// TIA Portal V16 program export: 0 tag tables, 14 data types, 2 data blocks, 1 code blocks (in call order from the OBs), 2 instance data blocks

TYPE "ConfigIF_MPLC_to_Plant"
// stored: IsFailsafeCompliant false
   STRUCT
      Spare_1 { ExternalAccessible := 'False'; ExternalVisible := 'False'; ExternalWritable := 'False'} : Word;   // Machine Features (refer to the Standard Machine Configuration Data)
      Machine_Product_ID { ExternalAccessible := 'False'; ExternalVisible := 'False'; ExternalWritable := 'False'} : Byte;   // Machine Product ID (refer to the Standard Machine Configuration Data)
      Machine_SortFraction { ExternalAccessible := 'False'; ExternalVisible := 'False'; ExternalWritable := 'False'} : Byte;   // Machine Sort Fraction (refer to the Standard Machine Configuration Data)
      Machine_Function { ExternalAccessible := 'False'; ExternalVisible := 'False'; ExternalWritable := 'False'} : Byte;   // Machine Function (refer to the Standard Machine Configuration Data)
      Machine_Cluster_ID { ExternalAccessible := 'False'; ExternalVisible := 'False'; ExternalWritable := 'False'} : Byte;   // Machine Cluster number (0-255)
      Machine_Cluster_Configuration { ExternalAccessible := 'False'; ExternalVisible := 'False'; ExternalWritable := 'False'} : Word;   // Machine Cluster Configuration (refer to the Standard Machine Configuration Data)
      PCS_PrimaryProtocol { ExternalAccessible := 'False'; ExternalVisible := 'False'; ExternalWritable := 'False'} : Byte;   // Primary Plant communication Protocol (Refer to Standard Machine Configuration Document)
      PCS_SecondaryProtocol { ExternalAccessible := 'False'; ExternalVisible := 'False'; ExternalWritable := 'False'} : Byte;   // Secondary Plant communication Protocol (Refer to Standard Machine Configuration Document)
      Hardware_Configuration_ID { ExternalAccessible := 'False'; ExternalVisible := 'False'; ExternalWritable := 'False'} : Byte;   // Machine PLC hardware configuration option (0-255)
      OPC_UA_ControlClient { ExternalAccessible := 'False'; ExternalVisible := 'False'; ExternalWritable := 'False'} : Bool;   // 0= Control Client Disabled; 1=Control Client Enabled
      OPC_UA_ViewClient_1 { ExternalAccessible := 'False'; ExternalVisible := 'False'; ExternalWritable := 'False'} : Bool;   // 0= View Client 1 Disabled; 1=View Client 1 Enabled
      OPC_UA_ViewClient_2 { ExternalAccessible := 'False'; ExternalVisible := 'False'; ExternalWritable := 'False'} : Bool;   // 0= View Client 2 Disabled; 1=View Client 2 Enabled
      OPC_UA_ViewClient_3 { ExternalAccessible := 'False'; ExternalVisible := 'False'; ExternalWritable := 'False'} : Bool;   // 0= View Client 3 Disabled; 1=View Client 3 Enabled
      Spare11_4 { ExternalAccessible := 'False'; ExternalVisible := 'False'; ExternalWritable := 'False'} : Bool;   // Reserved spare
      Spare11_5 { ExternalAccessible := 'False'; ExternalVisible := 'False'; ExternalWritable := 'False'} : Bool;   // Reserved spare
      Spare11_6 { ExternalAccessible := 'False'; ExternalVisible := 'False'; ExternalWritable := 'False'} : Bool;   // Reserved spare
      Spare11_7 { ExternalAccessible := 'False'; ExternalVisible := 'False'; ExternalWritable := 'False'} : Bool;   // Reserved spare
      Machine_IP_Address { ExternalAccessible := 'False'; ExternalVisible := 'False'; ExternalWritable := 'False'} : Array[1..4] of Byte;   // Machine PLC IP address (xx-xx-xx-xx)
      Machine_TCP_Port { ExternalAccessible := 'False'; ExternalVisible := 'False'; ExternalWritable := 'False'} : Int;   // Machine PLC TCP port number (2010-5000)
      Machine_TSAP { ExternalAccessible := 'False'; ExternalVisible := 'False'; ExternalWritable := 'False'} : Array[1..16] of Byte;   // Machine PLC TSAP (string containing Machine to 16 x ASCII characters)
      Machine_MAC_Address { ExternalAccessible := 'False'; ExternalVisible := 'False'; ExternalWritable := 'False'} : Array[0..5] of Byte;   // Machine PLC MAC address (xx-xx-xx-xx-xx-xx)
      Plant_Connection_ID { ExternalAccessible := 'False'; ExternalVisible := 'False'; ExternalWritable := 'False'} : Int;   // Plant PLC connection reference (1-65535)
      Spare { ExternalAccessible := 'False'; ExternalVisible := 'False'; ExternalWritable := 'False'} : Int;   // Reserved spare
      NTP_Server_IP_Address { ExternalAccessible := 'False'; ExternalVisible := 'False'; ExternalWritable := 'False'} : Array[1..4] of Byte;   // NTP Time Server Address (xx-xx-xx-xx)
      Last_PCS_Config_Hours { ExternalAccessible := 'False'; ExternalVisible := 'False'; ExternalWritable := 'False'} : Byte;   // Last configuration date/time recorded on the PLC after PCS config request from OTI or Plant. OTI/SCADA username transferred by PLC (depending on the config source)
      Last_PCS_Config_Minutes { ExternalAccessible := 'False'; ExternalVisible := 'False'; ExternalWritable := 'False'} : Byte;   // As above
      Last_PCS_Config_Century { ExternalAccessible := 'False'; ExternalVisible := 'False'; ExternalWritable := 'False'} : Byte;   // As above
      Last_PCS_Config_Year { ExternalAccessible := 'False'; ExternalVisible := 'False'; ExternalWritable := 'False'} : Byte;   // As above
      Last_PCS_Config_Month { ExternalAccessible := 'False'; ExternalVisible := 'False'; ExternalWritable := 'False'} : Byte;   // As above
      Last_PCS_Config_Day { ExternalAccessible := 'False'; ExternalVisible := 'False'; ExternalWritable := 'False'} : Byte;   // As above
      UserName { ExternalAccessible := 'False'; ExternalVisible := 'False'; ExternalWritable := 'False'} : Array[0..7] of Byte;   // Name of user (SCADA or OTI), who performed PCS configuration
      PCS_Config_Source { ExternalAccessible := 'False'; ExternalVisible := 'False'; ExternalWritable := 'False'} : Byte;   // PCS Configuration source: 0 - None; 1 - OTI; 2 - Plant
      OPC_UA_ControlClient_Active { ExternalAccessible := 'False'; ExternalVisible := 'False'; ExternalWritable := 'False'} : Bool;   // 1=OPC-UA ControlClient Active; 0=OPC-UA ControlClient Inactive
      OPC_UA_ViewClient_1_Active { ExternalAccessible := 'False'; ExternalVisible := 'False'; ExternalWritable := 'False'} : Bool;   // 1=OPC-UA ViewClient_1 Active; 0=OPC-UA ViewClient_1 Inactive
      OPC_UA_ViewClient_2_Active { ExternalAccessible := 'False'; ExternalVisible := 'False'; ExternalWritable := 'False'} : Bool;   // 1=OPC-UA ViewClient_2 Active; 0=OPC-UA ViewClient_2 Inactive
      OPC_UA_ViewClient_3_Active { ExternalAccessible := 'False'; ExternalVisible := 'False'; ExternalWritable := 'False'} : Bool;   // 1=OPC-UA ViewClient_3 Active; 0=OPC-UA ViewClient_3 Inactive
      Spare63_4 { ExternalAccessible := 'False'; ExternalVisible := 'False'; ExternalWritable := 'False'} : Bool;   // Reserved spare
      Spare63_5 { ExternalAccessible := 'False'; ExternalVisible := 'False'; ExternalWritable := 'False'} : Bool;   // Reserved spare
      Primary_Protocol_Comms_OK { ExternalAccessible := 'False'; ExternalVisible := 'False'; ExternalWritable := 'False'} : Bool;   // Plant Control Network Communication Status (0=Error; 1=OK)
      Secondary_Protocol_Comms_OK { ExternalAccessible := 'False'; ExternalVisible := 'False'; ExternalWritable := 'False'} : Bool;   // Plant SMachineervision Network Communication Status (0=Error; 1=OK)
      OPC_UA_PortNumber { ExternalAccessible := 'False'; ExternalVisible := 'False'; ExternalWritable := 'False'} : UInt;   // Machine- configured OPC-UA port
      Profibus_Address { ExternalAccessible := 'False'; ExternalVisible := 'False'; ExternalWritable := 'False'} : Byte;   // Machine- configured Profibus Address
      Spare67 { ExternalAccessible := 'False'; ExternalVisible := 'False'; ExternalWritable := 'False'} : Byte;   // Reserved spare
      Spare68 { ExternalAccessible := 'False'; ExternalVisible := 'False'; ExternalWritable := 'False'} : Byte;   // Reserved spare
      Spare69 { ExternalAccessible := 'False'; ExternalVisible := 'False'; ExternalWritable := 'False'} : Byte;   // Reserved spare
      Spare70 { ExternalAccessible := 'False'; ExternalVisible := 'False'; ExternalWritable := 'False'} : Byte;   // Reserved spare
      Spare71 { ExternalAccessible := 'False'; ExternalVisible := 'False'; ExternalWritable := 'False'} : Byte;   // Reserved spare
      Spare72 { ExternalAccessible := 'False'; ExternalVisible := 'False'; ExternalWritable := 'False'} : Byte;   // Reserved spare
      Spare73 { ExternalAccessible := 'False'; ExternalVisible := 'False'; ExternalWritable := 'False'} : Byte;   // Reserved spare
      Spare74 { ExternalAccessible := 'False'; ExternalVisible := 'False'; ExternalWritable := 'False'} : Byte;   // Reserved spare
      Spare75 { ExternalAccessible := 'False'; ExternalVisible := 'False'; ExternalWritable := 'False'} : Byte;   // Reserved spare
      Spare76 { ExternalAccessible := 'False'; ExternalVisible := 'False'; ExternalWritable := 'False'} : Byte;   // Reserved spare
      Spare77 { ExternalAccessible := 'False'; ExternalVisible := 'False'; ExternalWritable := 'False'} : Byte;   // Reserved spare
      Spare78 { ExternalAccessible := 'False'; ExternalVisible := 'False'; ExternalWritable := 'False'} : Byte;   // Reserved spare
      Spare79 { ExternalAccessible := 'False'; ExternalVisible := 'False'; ExternalWritable := 'False'} : Byte;   // Reserved spare
      Spare80 { ExternalAccessible := 'False'; ExternalVisible := 'False'; ExternalWritable := 'False'} : Byte;   // Reserved spare
      Spare81 { ExternalAccessible := 'False'; ExternalVisible := 'False'; ExternalWritable := 'False'} : Byte;   // Reserved spare
      Spare82 { ExternalAccessible := 'False'; ExternalVisible := 'False'; ExternalWritable := 'False'} : Byte;   // Reserved spare
      Spare83 { ExternalAccessible := 'False'; ExternalVisible := 'False'; ExternalWritable := 'False'} : Byte;   // Reserved spare
      Spare84 { ExternalAccessible := 'False'; ExternalVisible := 'False'; ExternalWritable := 'False'} : Byte;   // Reserved spare
      Spare85 { ExternalAccessible := 'False'; ExternalVisible := 'False'; ExternalWritable := 'False'} : Byte;   // Reserved spare
      Spare86 { ExternalAccessible := 'False'; ExternalVisible := 'False'; ExternalWritable := 'False'} : Byte;   // Reserved spare
      Spare87 { ExternalAccessible := 'False'; ExternalVisible := 'False'; ExternalWritable := 'False'} : Byte;   // Reserved spare
      Spare88 { ExternalAccessible := 'False'; ExternalVisible := 'False'; ExternalWritable := 'False'} : Byte;   // Reserved spare
      Spare89 { ExternalAccessible := 'False'; ExternalVisible := 'False'; ExternalWritable := 'False'} : Byte;   // Reserved spare
      Machine_Features { ExternalAccessible := 'False'; ExternalVisible := 'False'; ExternalWritable := 'False'} : DWord;   // Machine Features (refer to the Standard Machine Configuration Data)
      Machine_Features_Mask { ExternalAccessible := 'False'; ExternalVisible := 'False'; ExternalWritable := 'False'} : DWord;   // Machine Features Mask (refer to the Standard Machine Configuration Data)
      OTI_CheckCycle_Override_Control_State { ExternalAccessible := 'False'; ExternalVisible := 'False'; ExternalWritable := 'False'} : Bool;   // 1 = 'Override Checkercycle' control on OTI Disabled
      OTI_Configuration_Control_Status { ExternalAccessible := 'False'; ExternalVisible := 'False'; ExternalWritable := 'False'} : Bool;   // 1 = OTI PCS Configuration Machinedate button disabled
      OTI_PCS_Config { ExternalAccessible := 'False'; ExternalVisible := 'False'; ExternalWritable := 'False'} : Bool;   // Configuration pulse from OTI (pulsed for 1sec)
      OTI_Authentication_Mode { ExternalAccessible := 'False'; ExternalVisible := 'False'; ExternalWritable := 'False'} : Bool;   // Machine user authentication mode (0=password; 1= biometrics)
      Machine_Init { ExternalAccessible := 'False'; ExternalVisible := 'False'; ExternalWritable := 'False'} : Bool;   // PLC IP Address /HW Config Machinedate pulse (pulsed for 1sec)
      OTI_Ej_Sense_Feedback_Control_State { ExternalAccessible := 'False'; ExternalVisible := 'False'; ExternalWritable := 'False'} : Bool;   // 1 = 'Override Ejector Sense Feedback Alarms' on OTI disabled
      Spare98_6 { ExternalAccessible := 'False'; ExternalVisible := 'False'; ExternalWritable := 'False'} : Bool;   // Reserved spare
      TimeSync_Source { ExternalAccessible := 'False'; ExternalVisible := 'False'; ExternalWritable := 'False'} : Bool;   // Time Synchronization Source (0=NTP Server; 1= Interface DB)
      Spare99_0 { ExternalAccessible := 'False'; ExternalVisible := 'False'; ExternalWritable := 'False'} : Bool;   // Reserved spare
      Spare99_1 { ExternalAccessible := 'False'; ExternalVisible := 'False'; ExternalWritable := 'False'} : Bool;   // Reserved spare
      Spare99_2 { ExternalAccessible := 'False'; ExternalVisible := 'False'; ExternalWritable := 'False'} : Bool;   // Reserved spare
      Spare99_3 { ExternalAccessible := 'False'; ExternalVisible := 'False'; ExternalWritable := 'False'} : Bool;   // Reserved spare
      Spare99_4 { ExternalAccessible := 'False'; ExternalVisible := 'False'; ExternalWritable := 'False'} : Bool;   // Reserved spare
      Spare99_5 { ExternalAccessible := 'False'; ExternalVisible := 'False'; ExternalWritable := 'False'} : Bool;   // Reserved spare
      Spare99_6 { ExternalAccessible := 'False'; ExternalVisible := 'False'; ExternalWritable := 'False'} : Bool;   // Reserved spare
      PCS_Config_Machinedate_Done { ExternalAccessible := 'False'; ExternalVisible := 'False'; ExternalWritable := 'False'} : Bool;   // 1 sec Confirmation pulse – configuration date, time and username recorded in the event log
   END_STRUCT;
END_TYPE

TYPE "ConfigIF_Plant_to_MPLC"
// stored: IsFailsafeCompliant false
   STRUCT
      Plant_ID { ExternalAccessible := 'False'; ExternalVisible := 'False'; ExternalWritable := 'False'} : Byte;   // Plant location code (Refer to Standard Machine Configuration Document)
      Area_ID { ExternalAccessible := 'False'; ExternalVisible := 'False'; ExternalWritable := 'False'} : Byte;   // Plant Area code (Refer to Standard Machine Configuration Document)
      Spare2 { ExternalAccessible := 'False'; ExternalVisible := 'False'; ExternalWritable := 'False'} : Byte;   // Reserved spare
      Machine_SortFraction { ExternalAccessible := 'False'; ExternalVisible := 'False'; ExternalWritable := 'False'} : Byte;   // Machine Sort Fraction (Refer to Standard Machine Configuration Document)
      Machine_Function { ExternalAccessible := 'False'; ExternalVisible := 'False'; ExternalWritable := 'False'} : Byte;   // Machine Function (Refer to Standard Machine Configuration Document)
      Machine_Cluster_ID { ExternalAccessible := 'False'; ExternalVisible := 'False'; ExternalWritable := 'False'} : Byte;   // Machine Cluster number (0-255)
      Machine_Cluster_Configuration { ExternalAccessible := 'False'; ExternalVisible := 'False'; ExternalWritable := 'False'} : UInt;   // Machine Cluster Configuration (Maximum of 4 Machine Functions)
      Station_Name { ExternalAccessible := 'False'; ExternalVisible := 'False'; ExternalWritable := 'False'} : Array[0..15] of Byte;   // Machine Station name (string containing 16 x ASCII characters)
      PCS_Type { ExternalAccessible := 'False'; ExternalVisible := 'False'; ExternalWritable := 'False'} : Byte;   // SCADA/Plant control system type
      PCS_SecondaryProtocol { ExternalAccessible := 'False'; ExternalVisible := 'False'; ExternalWritable := 'False'} : Byte;   // Secondary Plant communication Protocol (Refer to Standard Machine Configuration Document)
      Plant_PLC_Type { ExternalAccessible := 'False'; ExternalVisible := 'False'; ExternalWritable := 'False'} : Byte;   // Plant PLC type and model
      OPCUA_ControlClient { ExternalAccessible := 'False'; ExternalVisible := 'False'; ExternalWritable := 'False'} : Bool;   // 0= Control Client Disabled; 1=Control Client Enabled
      OPCUA_ViewClient_1 { ExternalAccessible := 'False'; ExternalVisible := 'False'; ExternalWritable := 'False'} : Bool;   // 0= View Client 1 Disabled; 1=View Client 1 Enabled
      OPCUA_ViewClient_2 { ExternalAccessible := 'False'; ExternalVisible := 'False'; ExternalWritable := 'False'} : Bool;   // 0= View Client 2 Disabled; 1=View Client 2 Enabled
      OPCUA_ViewClient_3 { ExternalAccessible := 'False'; ExternalVisible := 'False'; ExternalWritable := 'False'} : Bool;   // 0= View Client 3 Disabled; 1=View Client 3 Enabled
      Spare27_4 { ExternalAccessible := 'False'; ExternalVisible := 'False'; ExternalWritable := 'False'} : Bool;   // Reserved spare
      Spare27_5 { ExternalAccessible := 'False'; ExternalVisible := 'False'; ExternalWritable := 'False'} : Bool;   // Reserved spare
      Spare27_6 { ExternalAccessible := 'False'; ExternalVisible := 'False'; ExternalWritable := 'False'} : Bool;   // Reserved spare
      Spare27_7 { ExternalAccessible := 'False'; ExternalVisible := 'False'; ExternalWritable := 'False'} : Bool;   // Reserved spare
      Spare28_4 { ExternalAccessible := 'False'; ExternalVisible := 'False'; ExternalWritable := 'False'} : DWord;   // Reserved spare
      Spare32_4 { ExternalAccessible := 'False'; ExternalVisible := 'False'; ExternalWritable := 'False'} : DWord;   // Reserved spare
      Spare36_4 { ExternalAccessible := 'False'; ExternalVisible := 'False'; ExternalWritable := 'False'} : DWord;   // Reserved spare
      Plant_IP_Address { ExternalAccessible := 'False'; ExternalVisible := 'False'; ExternalWritable := 'False'} : Array[1..4] of Byte;   // Plant PLC IP address (xx-xx-xx-xx)
      Machine_Port_Number { ExternalAccessible := 'False'; ExternalVisible := 'False'; ExternalWritable := 'False'} : UInt;   // Machine PLC TCP port number (2010-5000)
      Plant_Port_Number { ExternalAccessible := 'False'; ExternalVisible := 'False'; ExternalWritable := 'False'} : UInt;   // Plant PLC TCP port number (2010-5000)
      Machine_TSAP { ExternalAccessible := 'False'; ExternalVisible := 'False'; ExternalWritable := 'False'} : Array[1..16] of Byte;   // Machine PLC TSAP (string containing Machine to 16 x ASCII characters)
      Plant_TSAP { ExternalAccessible := 'False'; ExternalVisible := 'False'; ExternalWritable := 'False'} : Array[1..16] of Byte;   // Plant PLC TSAP (string containing Machine to 16 x ASCII characters)
      Spare80_4 { ExternalAccessible := 'False'; ExternalVisible := 'False'; ExternalWritable := 'False'} : DWord;   // Reserved spare
      Spare84_2 { ExternalAccessible := 'False'; ExternalVisible := 'False'; ExternalWritable := 'False'} : Word;   // Reserved spare
      Plant_MAC_Address { ExternalAccessible := 'False'; ExternalVisible := 'False'; ExternalWritable := 'False'} : Array[0..5] of Byte;   // Plant PLC MAC address (xx-xx-xx-xx)
      PCS_Connection_ID { ExternalAccessible := 'False'; ExternalVisible := 'False'; ExternalWritable := 'False'} : UInt;   // Plant PLC connection reference (1-65535)
      NTP_Server_IP_Address { ExternalAccessible := 'False'; ExternalVisible := 'False'; ExternalWritable := 'False'} : Array[1..4] of Byte;   // NTP time server address (xx-xx-xx-xx)
      UserName { ExternalAccessible := 'False'; ExternalVisible := 'False'; ExternalWritable := 'False'} : Array[0..7] of Byte;   // SCADA login username (Machine to 8 ASCII characters)
      DataServer_IP_Address { ExternalAccessible := 'False'; ExternalVisible := 'False'; ExternalWritable := 'False'} : Array[1..4] of Byte;   // Shared Data Server IP Address (xx-xx-xx-xx)
      DataServer_Subnet_Mask { ExternalAccessible := 'False'; ExternalVisible := 'False'; ExternalWritable := 'False'} : Array[1..4] of Byte;   // Shared Data Server Subnet Mask (xx-xx-xx-xx)
      DNS_Server_Address { ExternalAccessible := 'False'; ExternalVisible := 'False'; ExternalWritable := 'False'} : Array[1..4] of Byte;   // Domain Name System IP Address (xx-xx-xx-xx)
      Spare118 { ExternalAccessible := 'False'; ExternalVisible := 'False'; ExternalWritable := 'False'} : Byte;   // Reserved spare
      Spare119 { ExternalAccessible := 'False'; ExternalVisible := 'False'; ExternalWritable := 'False'} : Byte;   // Reserved spare
      Spare120 { ExternalAccessible := 'False'; ExternalVisible := 'False'; ExternalWritable := 'False'} : Byte;   // Reserved spare
      Spare121 { ExternalAccessible := 'False'; ExternalVisible := 'False'; ExternalWritable := 'False'} : Byte;   // Reserved spare
      Spare122 { ExternalAccessible := 'False'; ExternalVisible := 'False'; ExternalWritable := 'False'} : Byte;   // Reserved spare
      Spare123 { ExternalAccessible := 'False'; ExternalVisible := 'False'; ExternalWritable := 'False'} : Byte;   // Reserved spare
      Spare124 { ExternalAccessible := 'False'; ExternalVisible := 'False'; ExternalWritable := 'False'} : Byte;   // Reserved spare
      Spare125 { ExternalAccessible := 'False'; ExternalVisible := 'False'; ExternalWritable := 'False'} : Byte;   // Reserved spare
      Spare126 { ExternalAccessible := 'False'; ExternalVisible := 'False'; ExternalWritable := 'False'} : Byte;   // Reserved spare
      Spare127 { ExternalAccessible := 'False'; ExternalVisible := 'False'; ExternalWritable := 'False'} : Byte;   // Reserved spare
      Spare128 { ExternalAccessible := 'False'; ExternalVisible := 'False'; ExternalWritable := 'False'} : Byte;   // Reserved spare
      Spare129 { ExternalAccessible := 'False'; ExternalVisible := 'False'; ExternalWritable := 'False'} : Byte;   // Reserved spare
      Spare130 { ExternalAccessible := 'False'; ExternalVisible := 'False'; ExternalWritable := 'False'} : Byte;   // Reserved spare
      Spare131 { ExternalAccessible := 'False'; ExternalVisible := 'False'; ExternalWritable := 'False'} : Byte;   // Reserved spare
      Spare132 { ExternalAccessible := 'False'; ExternalVisible := 'False'; ExternalWritable := 'False'} : Byte;   // Reserved spare
      Spare133 { ExternalAccessible := 'False'; ExternalVisible := 'False'; ExternalWritable := 'False'} : Byte;   // Reserved spare
      Spare134 { ExternalAccessible := 'False'; ExternalVisible := 'False'; ExternalWritable := 'False'} : Byte;   // Reserved spare
      Spare135 { ExternalAccessible := 'False'; ExternalVisible := 'False'; ExternalWritable := 'False'} : Byte;   // Reserved spare
      Spare136 { ExternalAccessible := 'False'; ExternalVisible := 'False'; ExternalWritable := 'False'} : Byte;   // Reserved spare
      Spare137 { ExternalAccessible := 'False'; ExternalVisible := 'False'; ExternalWritable := 'False'} : Byte;   // Reserved spare
      Spare138 { ExternalAccessible := 'False'; ExternalVisible := 'False'; ExternalWritable := 'False'} : Byte;   // Reserved spare
      Spare139 { ExternalAccessible := 'False'; ExternalVisible := 'False'; ExternalWritable := 'False'} : Byte;   // Reserved spare
      Spare140 { ExternalAccessible := 'False'; ExternalVisible := 'False'; ExternalWritable := 'False'} : Byte;   // Reserved spare
      Spare141 { ExternalAccessible := 'False'; ExternalVisible := 'False'; ExternalWritable := 'False'} : Byte;   // Reserved spare
      Spare142 { ExternalAccessible := 'False'; ExternalVisible := 'False'; ExternalWritable := 'False'} : Byte;   // Reserved spare
      Spare143 { ExternalAccessible := 'False'; ExternalVisible := 'False'; ExternalWritable := 'False'} : Byte;   // Reserved spare
      Spare144 { ExternalAccessible := 'False'; ExternalVisible := 'False'; ExternalWritable := 'False'} : Byte;   // Reserved spare
      Spare145 { ExternalAccessible := 'False'; ExternalVisible := 'False'; ExternalWritable := 'False'} : Byte;   // Reserved spare
      "Checker Cycle Override Disable" { ExternalAccessible := 'False'; ExternalVisible := 'False'; ExternalWritable := 'False'} : Bool;   // Disable 'Override Checkercycle' control located on the OTI
      Ejector_Feedback_Override_Disable { ExternalAccessible := 'False'; ExternalVisible := 'False'; ExternalWritable := 'False'} : Bool;   // Disable 'Ejector Sense Feedback Override' control located on the OTI
      Spare146_2 { ExternalAccessible := 'False'; ExternalVisible := 'False'; ExternalWritable := 'False'} : Bool;   // Reserved spare
      Spare146_3 { ExternalAccessible := 'False'; ExternalVisible := 'False'; ExternalWritable := 'False'} : Bool;   // Reserved spare
      Spare146_4 { ExternalAccessible := 'False'; ExternalVisible := 'False'; ExternalWritable := 'False'} : Bool;   // Reserved spare
      Spare146_5 { ExternalAccessible := 'False'; ExternalVisible := 'False'; ExternalWritable := 'False'} : Bool;   // Reserved spare
      Spare146_6 { ExternalAccessible := 'False'; ExternalVisible := 'False'; ExternalWritable := 'False'} : Bool;   // Reserved spare
      Spare146_7 { ExternalAccessible := 'False'; ExternalVisible := 'False'; ExternalWritable := 'False'} : Bool;   // Reserved spare
      Spare147 { ExternalAccessible := 'False'; ExternalVisible := 'False'; ExternalWritable := 'False'} : Byte;   // Reserved spare
      Spare148_0 { ExternalAccessible := 'False'; ExternalVisible := 'False'; ExternalWritable := 'False'} : Bool;   // Reserved spare
      OTI_Configuration_Control { ExternalAccessible := 'False'; ExternalVisible := 'False'; ExternalWritable := 'False'} : Bool;   // Enable/disable OTI PCS configuration controls
      Plant_PCS_Config { ExternalAccessible := 'False'; ExternalVisible := 'False'; ExternalWritable := 'False'} : Bool;   // Plant PCS Configuration request
      Authentication_Mode { ExternalAccessible := 'False'; ExternalVisible := 'False'; ExternalWritable := 'False'} : Bool;   // Machine user authentication mode (0=password; 1= biometrics)
      Spare148_4 { ExternalAccessible := 'False'; ExternalVisible := 'False'; ExternalWritable := 'False'} : Bool;   // Reserved spare
      Spare148_5 { ExternalAccessible := 'False'; ExternalVisible := 'False'; ExternalWritable := 'False'} : Bool;   // Reserved spare
      Secondary_Protocol_Disable { ExternalAccessible := 'False'; ExternalVisible := 'False'; ExternalWritable := 'False'} : Bool;   // 1=Disable Secondary Protocol
      TimeSync_Source { ExternalAccessible := 'False'; ExternalVisible := 'False'; ExternalWritable := 'False'} : Bool;   // Time Synchronization Source (0=NTP Server; 1= Interface DB)
      Spare149_0 { ExternalAccessible := 'False'; ExternalVisible := 'False'; ExternalWritable := 'False'} : Bool;   // Reserved spare
      Spare149_1 { ExternalAccessible := 'False'; ExternalVisible := 'False'; ExternalWritable := 'False'} : Bool;   // Reserved spare
      Spare149_2 { ExternalAccessible := 'False'; ExternalVisible := 'False'; ExternalWritable := 'False'} : Bool;   // Reserved spare
      Spare149_3 { ExternalAccessible := 'False'; ExternalVisible := 'False'; ExternalWritable := 'False'} : Bool;   // Reserved spare
      Spare149_4 { ExternalAccessible := 'False'; ExternalVisible := 'False'; ExternalWritable := 'False'} : Bool;   // Reserved spare
      Spare149_5 { ExternalAccessible := 'False'; ExternalVisible := 'False'; ExternalWritable := 'False'} : Bool;   // Reserved spare
      Spare149_6 { ExternalAccessible := 'False'; ExternalVisible := 'False'; ExternalWritable := 'False'} : Bool;   // Reserved spare
      Spare149_7 { ExternalAccessible := 'False'; ExternalVisible := 'False'; ExternalWritable := 'False'} : Bool;   // Reserved spare
   END_STRUCT;
END_TYPE

TYPE "PLANT_SEQ_STATE"
// stored: IsFailsafeCompliant false
   STRUCT
      Ready { ExternalVisible := 'False'; ExternalWritable := 'False'} : Bool;   // Ready for Control
      Safety_Interlock { ExternalVisible := 'False'; ExternalWritable := 'False'} : Bool;   // Safety Interlock
      Process_Interlock { ExternalVisible := 'False'; ExternalWritable := 'False'} : Bool;   // Process Interlock
      Hold { ExternalVisible := 'False'; ExternalWritable := 'False'} : Bool;   // Hold State
      Wait { ExternalVisible := 'False'; ExternalWritable := 'False'} : Bool;   // Wait State
      Reserved0 { ExternalVisible := 'False'; ExternalWritable := 'False'} : Bool;   // Reserved spare
      Manual { ExternalVisible := 'False'; ExternalWritable := 'False'} : Bool;   // 0 = Machine Auto, 1 = Machine Manual
      Alarm { ExternalVisible := 'False'; ExternalWritable := 'False'} : Bool;   // Alarm State
      Maintenance { ExternalVisible := 'False'; ExternalWritable := 'False'} : Bool;   // 1 = Maintenance
      Up_Stream_Interlock { ExternalVisible := 'False'; ExternalWritable := 'False'} : Bool;   // UP Stream Interlock Set by Machine
      Reserved1 { ExternalVisible := 'False'; ExternalWritable := 'False'} : Bool;   // Reserved spare
      Reserved2 { ExternalVisible := 'False'; ExternalWritable := 'False'} : Bool;   // Reserved spare
      Reserved3 { ExternalVisible := 'False'; ExternalWritable := 'False'} : Bool;   // Reserved spare
      Reserved4 { ExternalVisible := 'False'; ExternalWritable := 'False'} : Bool;   // Reserved spare
      MPLC_to_MC_Comms_Fail { ExternalVisible := 'False'; ExternalWritable := 'False'} : Bool;   // Machine PLC to Machine Controller communication has failed
      SOC_Plant_Control_Status { ExternalVisible := 'False'; ExternalWritable := 'False'} : Bool;   // SOC_ Plant Control Status, 0 = Supervised Operator Control, 1 = Plant
      Machine_Initialising { ExternalVisible := 'False'; ExternalWritable := 'False'} : Bool;   // Machine in Initialising State
      Machine_Ready { ExternalVisible := 'False'; ExternalWritable := 'False'} : Bool;   // Machine in Ready state
      Machine_Purging { ExternalVisible := 'False'; ExternalWritable := 'False'} : Bool;   // Machine in Purge state
      Machine_Display { ExternalVisible := 'False'; ExternalWritable := 'False'} : Bool;   // Machine in Display state
      Machine_Calibrating { ExternalVisible := 'False'; ExternalWritable := 'False'} : Bool;   // Machine in Calibrating state
      Machine_Checker_Cycle { ExternalVisible := 'False'; ExternalWritable := 'False'} : Bool;   // Machine in Checker Cycle state
      Machine_Processing_Ready { ExternalVisible := 'False'; ExternalWritable := 'False'} : Bool;   // Machine in Process Ready State
      Machine_Processing { ExternalVisible := 'False'; ExternalWritable := 'False'} : Bool;   // Machine in Process with Feed state
      Machine_Transition { ExternalVisible := 'False'; ExternalWritable := 'False'} : Bool;   // Machine in Transition state
      Reserved6 { ExternalVisible := 'False'; ExternalWritable := 'False'} : Bool;   // Reserved for additional state
      Machine_Alarm { ExternalVisible := 'False'; ExternalWritable := 'False'} : Bool;   // Machine in Alarm State
      Reserved7 { ExternalVisible := 'False'; ExternalWritable := 'False'} : Bool;   // Reserved spare
      Reserved8 { ExternalVisible := 'False'; ExternalWritable := 'False'} : Bool;   // Reserved spare
      Reserved9 { ExternalVisible := 'False'; ExternalWritable := 'False'} : Bool;   // Reserved spare
      Reserved10 { ExternalVisible := 'False'; ExternalWritable := 'False'} : Bool;   // Reserved spare
      Reserved11 { ExternalVisible := 'False'; ExternalWritable := 'False'} : Bool;   // Reserved spare
      Command_Conf_Gen { ExternalVisible := 'False'; ExternalWritable := 'False'} : Bool;   // General Command Confirmation Reporting
      Command_Failure { ExternalVisible := 'False'; ExternalWritable := 'False'} : Bool;   // Command Failure Reporting - Command did not execute on the Machine
      Command_Busy { ExternalVisible := 'False'; ExternalWritable := 'False'} : Bool;   // Command Busy Reporting - UP Busy processing Command
      Command_Conf_Rec_Save { ExternalVisible := 'False'; ExternalWritable := 'False'} : Bool;   // Command Confirmation Reporting - Recipe Save
      Command_Conf_Rec_Del { ExternalVisible := 'False'; ExternalWritable := 'False'} : Bool;   // Command Confirmation Reporting - Recipe Delete
      Command_Conf_Rec_Copy { ExternalVisible := 'False'; ExternalWritable := 'False'} : Bool;   // Command Confirmation Reporting - Recipe Copy
      Reserved12 { ExternalVisible := 'False'; ExternalWritable := 'False'} : Bool;   // Reserved spare
      Logon_Successful { ExternalVisible := 'False'; ExternalWritable := 'False'} : Bool;   // Command Confirmation Reporting - Logon OK
      Reserved13 { ExternalVisible := 'False'; ExternalWritable := 'False'} : Byte;   // Reserved spare
      Current_Recipe_Selected { ExternalVisible := 'False'; ExternalWritable := 'False'} : Byte;   // Feedback Indicating the Recipe Number Loaded onto the Machine
      HEARTBEAT_MPLC_PCS { ExternalVisible := 'False'; ExternalWritable := 'False'} : Byte;   // Heartbeat to Plant Controller
      Reserved14 { ExternalVisible := 'False'; ExternalWritable := 'False'} : Byte;   // Spare
      Primary_Process_Intlk_Ext { ExternalVisible := 'False'; ExternalWritable := 'False'} : Bool;   // Primary Process Interlock External
      Secndry_Process_Intlk_Ext { ExternalVisible := 'False'; ExternalWritable := 'False'} : Bool;   // Secondary Interlock External
      Safety_Interlock_Ext { ExternalVisible := 'False'; ExternalWritable := 'False'} : Bool;   // Safety Interlock Ext
      SOC_Request { ExternalVisible := 'False'; ExternalWritable := 'False'} : Bool;   // Supervised Operator Interface control request
      Reserved16 { ExternalVisible := 'False'; ExternalWritable := 'False'} : Bool;   // Spare
      Reserved17 { ExternalVisible := 'False'; ExternalWritable := 'False'} : Bool;   // Spare
      Reserved18 { ExternalVisible := 'False'; ExternalWritable := 'False'} : Bool;   // Spare
      Reserved19 { ExternalVisible := 'False'; ExternalWritable := 'False'} : Bool;   // Spare
   END_STRUCT;
END_TYPE

TYPE "RTC"
// stored: IsFailsafeCompliant false
   STRUCT
      CLK_YEAR { ExternalAccessible := 'False'; ExternalVisible := 'False'; ExternalWritable := 'False'} : USInt;
      CLK_MONTH { ExternalAccessible := 'False'; ExternalVisible := 'False'; ExternalWritable := 'False'} : USInt;
      CLK_DAY { ExternalAccessible := 'False'; ExternalVisible := 'False'; ExternalWritable := 'False'} : USInt;
      CLK_HOUR { ExternalAccessible := 'False'; ExternalVisible := 'False'; ExternalWritable := 'False'} : USInt;
      CLK_MINUTE { ExternalAccessible := 'False'; ExternalVisible := 'False'; ExternalWritable := 'False'} : USInt;
      CLK_SECOND { ExternalAccessible := 'False'; ExternalVisible := 'False'; ExternalWritable := 'False'} : USInt;
   END_STRUCT;
END_TYPE

TYPE "118MK2_Bit_Commands"
// stored: IsFailsafeCompliant false
   STRUCT
      Start_M_PCS { ExternalAccessible := 'False'; ExternalVisible := 'False'; ExternalWritable := 'False'} : Bool;
      Stop_M_PCS { ExternalAccessible := 'False'; ExternalVisible := 'False'; ExternalWritable := 'False'} : Bool;
      Start_Feeding_M_PCS { ExternalAccessible := 'False'; ExternalVisible := 'False'; ExternalWritable := 'False'} : Bool;
      Stop_Feeding_M_PCS { ExternalAccessible := 'False'; ExternalVisible := 'False'; ExternalWritable := 'False'} : Bool;
      Checker_Cycle_M_PCS { ExternalAccessible := 'False'; ExternalVisible := 'False'; ExternalWritable := 'False'} : Bool;
      Purge_M_PCS { ExternalAccessible := 'False'; ExternalVisible := 'False'; ExternalWritable := 'False'} : Bool;
      Acknowledge_Alarm_PCS { ExternalAccessible := 'False'; ExternalVisible := 'False'; ExternalWritable := 'False'} : Bool;
      Reset_Alarm_PCS { ExternalAccessible := 'False'; ExternalVisible := 'False'; ExternalWritable := 'False'} : Bool;
      Manual_Req_PCS { ExternalAccessible := 'False'; ExternalVisible := 'False'; ExternalWritable := 'False'} : Bool;
      Calibrate_M_PCS { ExternalAccessible := 'False'; ExternalVisible := 'False'; ExternalWritable := 'False'} : Bool;
      Display_M_PCS { ExternalAccessible := 'False'; ExternalVisible := 'False'; ExternalWritable := 'False'} : Bool;
      Save_As_Reference_PCS { ExternalAccessible := 'False'; ExternalVisible := 'False'; ExternalWritable := 'False'} : Bool;
      Save_Oper_Params_PCS { ExternalAccessible := 'False'; ExternalVisible := 'False'; ExternalWritable := 'False'} : Bool;
      Upd_Sys_DateTime_PCS { ExternalAccessible := 'False'; ExternalVisible := 'False'; ExternalWritable := 'False'} : Bool;
      Spare6 { ExternalAccessible := 'False'; ExternalVisible := 'False'; ExternalWritable := 'False'} : Bool;
      Spare7 { ExternalAccessible := 'False'; ExternalVisible := 'False'; ExternalWritable := 'False'} : Bool;
      Clr_LiHist_M_PCS { ExternalAccessible := 'False'; ExternalVisible := 'False'; ExternalWritable := 'False'} : Bool;
      Clr_Profile_M_PCS { ExternalAccessible := 'False'; ExternalVisible := 'False'; ExternalWritable := 'False'} : Bool;
      Clr_EjecErrHist_M_PCS { ExternalAccessible := 'False'; ExternalVisible := 'False'; ExternalWritable := 'False'} : Bool;
      Clr_EjecResProf_M_PCS { ExternalAccessible := 'False'; ExternalVisible := 'False'; ExternalWritable := 'False'} : Bool;
      Clr_CCCalData_M_PCS { ExternalAccessible := 'False'; ExternalVisible := 'False'; ExternalWritable := 'False'} : Bool;
      Spare8 { ExternalAccessible := 'False'; ExternalVisible := 'False'; ExternalWritable := 'False'} : Bool;
      Spare9 { ExternalAccessible := 'False'; ExternalVisible := 'False'; ExternalWritable := 'False'} : Bool;
      Spare10 { ExternalAccessible := 'False'; ExternalVisible := 'False'; ExternalWritable := 'False'} : Bool;
      Spare11 { ExternalAccessible := 'False'; ExternalVisible := 'False'; ExternalWritable := 'False'} : Bool;
      Spare12 { ExternalAccessible := 'False'; ExternalVisible := 'False'; ExternalWritable := 'False'} : Bool;
      Spare13 { ExternalAccessible := 'False'; ExternalVisible := 'False'; ExternalWritable := 'False'} : Bool;
      Spare14 { ExternalAccessible := 'False'; ExternalVisible := 'False'; ExternalWritable := 'False'} : Bool;
      Spare15 { ExternalAccessible := 'False'; ExternalVisible := 'False'; ExternalWritable := 'False'} : Bool;
      Spare16 { ExternalAccessible := 'False'; ExternalVisible := 'False'; ExternalWritable := 'False'} : Bool;
      Spare17 { ExternalAccessible := 'False'; ExternalVisible := 'False'; ExternalWritable := 'False'} : Bool;
      Spare18 { ExternalAccessible := 'False'; ExternalVisible := 'False'; ExternalWritable := 'False'} : Bool;
      Add_New_User_PCS { ExternalAccessible := 'False'; ExternalVisible := 'False'; ExternalWritable := 'False'} : Bool;
      Del_Select_User_PCS { ExternalAccessible := 'False'; ExternalVisible := 'False'; ExternalWritable := 'False'} : Bool;
      Logon_User_PCS { ExternalAccessible := 'False'; ExternalVisible := 'False'; ExternalWritable := 'False'} : Bool;
      LogOff_User_PCS { ExternalAccessible := 'False'; ExternalVisible := 'False'; ExternalWritable := 'False'} : Bool;
      Change_User_Pass_PCS { ExternalAccessible := 'False'; ExternalVisible := 'False'; ExternalWritable := 'False'} : Bool;
      Lookup_User_PCS { ExternalAccessible := 'False'; ExternalVisible := 'False'; ExternalWritable := 'False'} : Bool;
      Spare19 { ExternalAccessible := 'False'; ExternalVisible := 'False'; ExternalWritable := 'False'} : Bool;
      Spare20 { ExternalAccessible := 'False'; ExternalVisible := 'False'; ExternalWritable := 'False'} : Bool;
      Start_A_PCS { ExternalAccessible := 'False'; ExternalVisible := 'False'; ExternalWritable := 'False'} : Bool;
      Stop_A_PCS { ExternalAccessible := 'False'; ExternalVisible := 'False'; ExternalWritable := 'False'} : Bool;
      Start_Feeding_A_PCS { ExternalAccessible := 'False'; ExternalVisible := 'False'; ExternalWritable := 'False'} : Bool;
      Stop_Feeding_A_PCS { ExternalAccessible := 'False'; ExternalVisible := 'False'; ExternalWritable := 'False'} : Bool;
      Checker_Cycle_A_PCS { ExternalAccessible := 'False'; ExternalVisible := 'False'; ExternalWritable := 'False'} : Bool;
      Purge_A_PCS { ExternalAccessible := 'False'; ExternalVisible := 'False'; ExternalWritable := 'False'} : Bool;
      Spare21 { ExternalAccessible := 'False'; ExternalVisible := 'False'; ExternalWritable := 'False'} : Bool;
      Spare22 { ExternalAccessible := 'False'; ExternalVisible := 'False'; ExternalWritable := 'False'} : Bool;
      Save_Recipe { ExternalAccessible := 'False'; ExternalVisible := 'False'; ExternalWritable := 'False'} : Bool;
      Delete_Recipe { ExternalAccessible := 'False'; ExternalVisible := 'False'; ExternalWritable := 'False'} : Bool;
      Copy_Recipe { ExternalAccessible := 'False'; ExternalVisible := 'False'; ExternalWritable := 'False'} : Bool;
      Spare23 { ExternalAccessible := 'False'; ExternalVisible := 'False'; ExternalWritable := 'False'} : Bool;
      Spare24 { ExternalAccessible := 'False'; ExternalVisible := 'False'; ExternalWritable := 'False'} : Bool;
      Spare25 { ExternalAccessible := 'False'; ExternalVisible := 'False'; ExternalWritable := 'False'} : Bool;
      Spare26 { ExternalAccessible := 'False'; ExternalVisible := 'False'; ExternalWritable := 'False'} : Bool;
      Spare27 { ExternalAccessible := 'False'; ExternalVisible := 'False'; ExternalWritable := 'False'} : Bool;
      Remote_DSInlk_PCS { ExternalAccessible := 'False'; ExternalVisible := 'False'; ExternalWritable := 'False'} : Bool;
      Remote_SpareCMD1_PCS { ExternalAccessible := 'False'; ExternalVisible := 'False'; ExternalWritable := 'False'} : Bool;
      Remote_SpareCMD2_PCS { ExternalAccessible := 'False'; ExternalVisible := 'False'; ExternalWritable := 'False'} : Bool;
      Remote_SpareCMD3_PCS { ExternalAccessible := 'False'; ExternalVisible := 'False'; ExternalWritable := 'False'} : Bool;
      Remote_SpareCMD4_PCS { ExternalAccessible := 'False'; ExternalVisible := 'False'; ExternalWritable := 'False'} : Bool;
      Remote_SpareCMD5_PCS { ExternalAccessible := 'False'; ExternalVisible := 'False'; ExternalWritable := 'False'} : Bool;
      Remote_SpareCMD6_PCS { ExternalAccessible := 'False'; ExternalVisible := 'False'; ExternalWritable := 'False'} : Bool;
      Remote_SpareCMD7_PCS { ExternalAccessible := 'False'; ExternalVisible := 'False'; ExternalWritable := 'False'} : Bool;
      SOC_Authorization { ExternalAccessible := 'False'; ExternalVisible := 'False'; ExternalWritable := 'False'} : Bool;
      SOC_Req_Acknowledge { ExternalAccessible := 'False'; ExternalVisible := 'False'; ExternalWritable := 'False'} : Bool;
      Spare30 { ExternalAccessible := 'False'; ExternalVisible := 'False'; ExternalWritable := 'False'} : Bool;
      Spare31 { ExternalAccessible := 'False'; ExternalVisible := 'False'; ExternalWritable := 'False'} : Bool;
      Spare32 { ExternalAccessible := 'False'; ExternalVisible := 'False'; ExternalWritable := 'False'} : Bool;
      Spare33 { ExternalAccessible := 'False'; ExternalVisible := 'False'; ExternalWritable := 'False'} : Bool;
      Spare34 { ExternalAccessible := 'False'; ExternalVisible := 'False'; ExternalWritable := 'False'} : Bool;
      Spare35 { ExternalAccessible := 'False'; ExternalVisible := 'False'; ExternalWritable := 'False'} : Bool;
      OPCUA_ControlClient { ExternalAccessible := 'False'; ExternalVisible := 'False'; ExternalWritable := 'False'} : Bool;
      "OPCUA_ViewClient _1" { ExternalAccessible := 'False'; ExternalVisible := 'False'; ExternalWritable := 'False'} : Bool;
      "OPCUA_ViewClient _2" { ExternalAccessible := 'False'; ExternalVisible := 'False'; ExternalWritable := 'False'} : Bool;
      "OPCUA_ViewClient _3" { ExternalAccessible := 'False'; ExternalVisible := 'False'; ExternalWritable := 'False'} : Bool;
      Spare27_4 { ExternalAccessible := 'False'; ExternalVisible := 'False'; ExternalWritable := 'False'} : Bool;
      Spare27_5 { ExternalAccessible := 'False'; ExternalVisible := 'False'; ExternalWritable := 'False'} : Bool;
      Spare27_6 { ExternalAccessible := 'False'; ExternalVisible := 'False'; ExternalWritable := 'False'} : Bool;
      Spare27_7 { ExternalAccessible := 'False'; ExternalVisible := 'False'; ExternalWritable := 'False'} : Bool;
      Override_CheckCycle_Disable { ExternalAccessible := 'False'; ExternalVisible := 'False'; ExternalWritable := 'False'} : Bool;
      OTI_Plant_Control { ExternalAccessible := 'False'; ExternalVisible := 'False'; ExternalWritable := 'False'} : Bool;
      Plant_PCS_Config { ExternalAccessible := 'False'; ExternalVisible := 'False'; ExternalWritable := 'False'} : Bool;
      Authentication_Mode { ExternalAccessible := 'False'; ExternalVisible := 'False'; ExternalWritable := 'False'} : Bool;
      Spare148_4 { ExternalAccessible := 'False'; ExternalVisible := 'False'; ExternalWritable := 'False'} : Bool;
      EjSense_Feedback_Override_Disable { ExternalAccessible := 'False'; ExternalVisible := 'False'; ExternalWritable := 'False'} : Bool;
      Secondary_Protocol_Disable { ExternalAccessible := 'False'; ExternalVisible := 'False'; ExternalWritable := 'False'} : Bool;
      Spare148_7 { ExternalAccessible := 'False'; ExternalVisible := 'False'; ExternalWritable := 'False'} : Bool;
      Spare149_0 { ExternalAccessible := 'False'; ExternalVisible := 'False'; ExternalWritable := 'False'} : Bool;
      Spare149_1 { ExternalAccessible := 'False'; ExternalVisible := 'False'; ExternalWritable := 'False'} : Bool;
      Spare149_2 { ExternalAccessible := 'False'; ExternalVisible := 'False'; ExternalWritable := 'False'} : Bool;
      Spare149_3 { ExternalAccessible := 'False'; ExternalVisible := 'False'; ExternalWritable := 'False'} : Bool;
      Spare149_4 { ExternalAccessible := 'False'; ExternalVisible := 'False'; ExternalWritable := 'False'} : Bool;
      Spare149_5 { ExternalAccessible := 'False'; ExternalVisible := 'False'; ExternalWritable := 'False'} : Bool;
      Spare149_6 { ExternalAccessible := 'False'; ExternalVisible := 'False'; ExternalWritable := 'False'} : Bool;
      Spare149_7 { ExternalAccessible := 'False'; ExternalVisible := 'False'; ExternalWritable := 'False'} : Bool;
   END_STRUCT;
END_TYPE

TYPE "118MK2_Command_Values"
// stored: IsFailsafeCompliant false
   STRUCT
      Start_CMD { ExternalAccessible := 'False'; ExternalVisible := 'False'; ExternalWritable := 'False'} : Byte := 1;   // Moves machine to Processing Ready state. Feeder is not started.
      Stop_CMD { ExternalAccessible := 'False'; ExternalVisible := 'False'; ExternalWritable := 'False'} : Byte := 2;   // Moves machine to Ready state. Hence also used to exit Display mode.
      Checker_Cycle_CMD { ExternalAccessible := 'False'; ExternalVisible := 'False'; ExternalWritable := 'False'} : Byte := 3;   // Initiates a Checker Cycle sequence
      Purge_CMD { ExternalAccessible := 'False'; ExternalVisible := 'False'; ExternalWritable := 'False'} : Byte := 4;   // Initiates a material purge sequence
      Calibrate_CMD { ExternalAccessible := 'False'; ExternalVisible := 'False'; ExternalWritable := 'False'} : Byte := 5;   // Automatically adjusts the PMT HV setpoints to achieve the desired calibration reference
      Display_CMD { ExternalAccessible := 'False'; ExternalVisible := 'False'; ExternalWritable := 'False'} : Byte := 6;   // Moves machine to Display state where blue and red channel data for all 8 channels is acquired every 250ms
      Acknowledge_Alarm_CMD { ExternalAccessible := 'False'; ExternalVisible := 'False'; ExternalWritable := 'False'} : Byte := 7;   // Acknowledges asserted alarms. Siren is deactivated
      Reset_Alarm_CMD { ExternalAccessible := 'False'; ExternalVisible := 'False'; ExternalWritable := 'False'} : Byte := 8;   // Resets asserted alarms
      Save_As_Reference_CMD { ExternalAccessible := 'False'; ExternalVisible := 'False'; ExternalWritable := 'False'} : Byte := 9;   // Saves the most recent calibration data for both the blue and red channels as the reference curve in the cRIO Controller non-volatile memory
      Start_Feeding_CMD { ExternalAccessible := 'False'; ExternalVisible := 'False'; ExternalWritable := 'False'} : Byte := 10;   // Starts the vibratory feeders
      Stop_Feeding_CMD { ExternalAccessible := 'False'; ExternalVisible := 'False'; ExternalWritable := 'False'} : Byte := 11;   // Stops the vibratory feeders
      Clr_LiHist_CMD { ExternalAccessible := 'False'; ExternalVisible := 'False'; ExternalWritable := 'False'} : Byte := 12;   // Clears Accepted, Rejected, Red and Blue-Red Ratio Luminescence Intensity Histograms
      Clr_Profile_CMD { ExternalAccessible := 'False'; ExternalVisible := 'False'; ExternalWritable := 'False'} : Byte := 13;   // Clears ejection, accepted & rejected profiles
      Clr_EjecErrHist_CMD { ExternalAccessible := 'False'; ExternalVisible := 'False'; ExternalWritable := 'False'} : Byte := 14;   // Resets all the data values in the Ejector error histograms to zero
      Clr_EjecResProf_CMD { ExternalAccessible := 'False'; ExternalVisible := 'False'; ExternalWritable := 'False'} : Byte := 15;   // Clears ejector delay response and ejector duration response profiles
      Clr_CCCalData_CMD { ExternalAccessible := 'False'; ExternalVisible := 'False'; ExternalWritable := 'False'} : Byte := 16;   // Clears Checker cycle calibration data blue & Checker cycle calibration data red profiles
      Add_New_User_CMD { ExternalAccessible := 'False'; ExternalVisible := 'False'; ExternalWritable := 'False'} : Byte := 25;   // Adds a new user based on username, password and access level specified, to the cRIO security lookup table
      Del_Selected_User_CMD { ExternalAccessible := 'False'; ExternalVisible := 'False'; ExternalWritable := 'False'} : Byte := 26;   // Delete the user specified by the current lookup table pointer, from the cRIO security lookup table
      Logon_User_CMD { ExternalAccessible := 'False'; ExternalVisible := 'False'; ExternalWritable := 'False'} : Byte := 27;   // Authorise user based on the specified username and password - the cRIO would return the appropriate access level
      Logoff_User_CMD { ExternalAccessible := 'False'; ExternalVisible := 'False'; ExternalWritable := 'False'} : Byte := 28;   // Log off user – the cRIO would return an access level of 0
      Cng_User_Password_CMD { ExternalAccessible := 'False'; ExternalVisible := 'False'; ExternalWritable := 'False'} : Byte := 29;   // Change password for currently logged on user as specified in “User password”
      Lookup_User_CMD { ExternalAccessible := 'False'; ExternalVisible := 'False'; ExternalWritable := 'False'} : Byte := 30;   // Retrieves the username and access level at the specified security lookup table pointer
      Save_Opr_Param_CMD { ExternalAccessible := 'False'; ExternalVisible := 'False'; ExternalWritable := 'False'} : Byte := 34;
      Upd_Sys_DateTime_CMD { ExternalAccessible := 'False'; ExternalVisible := 'False'; ExternalWritable := 'False'} : Byte := 39;
      SpareCmd_0 { ExternalAccessible := 'False'; ExternalVisible := 'False'; ExternalWritable := 'False'} : Byte;
      SpareCmd_1 { ExternalAccessible := 'False'; ExternalVisible := 'False'; ExternalWritable := 'False'} : Byte;
      SpareCmd_2 { ExternalAccessible := 'False'; ExternalVisible := 'False'; ExternalWritable := 'False'} : Byte;
      SpareCmd_3 { ExternalAccessible := 'False'; ExternalVisible := 'False'; ExternalWritable := 'False'} : Byte;
      SpareCmd_4 { ExternalAccessible := 'False'; ExternalVisible := 'False'; ExternalWritable := 'False'} : Byte;
      SpareCmd_5 { ExternalAccessible := 'False'; ExternalVisible := 'False'; ExternalWritable := 'False'} : Byte;
      SpareCmd_6 { ExternalAccessible := 'False'; ExternalVisible := 'False'; ExternalWritable := 'False'} : Byte;
      SpareCmd_7 { ExternalAccessible := 'False'; ExternalVisible := 'False'; ExternalWritable := 'False'} : Byte;
      SpareCmd_8 { ExternalAccessible := 'False'; ExternalVisible := 'False'; ExternalWritable := 'False'} : Byte;
      SpareCmd_9 { ExternalAccessible := 'False'; ExternalVisible := 'False'; ExternalWritable := 'False'} : Byte;
      SpareCmd_10 { ExternalAccessible := 'False'; ExternalVisible := 'False'; ExternalWritable := 'False'} : Byte;
      SpareCmd_11 { ExternalAccessible := 'False'; ExternalVisible := 'False'; ExternalWritable := 'False'} : Byte;
      SpareCmd_12 { ExternalAccessible := 'False'; ExternalVisible := 'False'; ExternalWritable := 'False'} : Byte;
      SpareCmd_13 { ExternalAccessible := 'False'; ExternalVisible := 'False'; ExternalWritable := 'False'} : Byte;
      SpareCmd_14 { ExternalAccessible := 'False'; ExternalVisible := 'False'; ExternalWritable := 'False'} : Byte;
      SpareCmd_15 { ExternalAccessible := 'False'; ExternalVisible := 'False'; ExternalWritable := 'False'} : Byte;
      SpareCmd_16 { ExternalAccessible := 'False'; ExternalVisible := 'False'; ExternalWritable := 'False'} : Byte;
      SpareCmd_17 { ExternalAccessible := 'False'; ExternalVisible := 'False'; ExternalWritable := 'False'} : Byte;
      SpareCmd_18 { ExternalAccessible := 'False'; ExternalVisible := 'False'; ExternalWritable := 'False'} : Byte;
      SpareCmd_19 { ExternalAccessible := 'False'; ExternalVisible := 'False'; ExternalWritable := 'False'} : Byte;
      SpareCmd_20 { ExternalAccessible := 'False'; ExternalVisible := 'False'; ExternalWritable := 'False'} : Byte;
      SpareCmd_21 { ExternalAccessible := 'False'; ExternalVisible := 'False'; ExternalWritable := 'False'} : Byte;
      SpareCmd_22 { ExternalAccessible := 'False'; ExternalVisible := 'False'; ExternalWritable := 'False'} : Byte;
      SpareCmd_23 { ExternalAccessible := 'False'; ExternalVisible := 'False'; ExternalWritable := 'False'} : Byte;
      SpareCmd_24 { ExternalAccessible := 'False'; ExternalVisible := 'False'; ExternalWritable := 'False'} : Byte;
      SpareCmd_25 { ExternalAccessible := 'False'; ExternalVisible := 'False'; ExternalWritable := 'False'} : Byte;
   END_STRUCT;
END_TYPE

TYPE "118MK2_PlantData"
// stored: IsFailsafeCompliant false
   STRUCT
      PLANT_TAG_NAME : Array[0..15] of Byte;   // Current plant tag name of the sorting module, 16 character string
      UP_MACHINE_NAME : Array[0..15] of Byte;   // Current manufacturer name of the sorting module – read from the cRIO Controller configuration, 16-character string
      COMMAND_ACK_S : Byte;   // Returns the (same) command value as an acknowledgement that the Real-time system has received the command.
      COMMAND_IN_PROG_S : Byte;   // Counts up as progress indicator – resets on completion
      INVALID_COMMAND_S : Bool;   // ‘1’ when an invalid command – cleared on next valid command.
      PARAM_OUT_OF_RANGE_S : Bool;   // ‘1’ when any requested parameter value is out of range.
      USER_ADDED_S : Bool;   // ‘1’ when a requested new user name was successfully added to the security lookup table.
      PASSWORD_CHANGED_S : Bool;   // ‘1’ when a requested password change was successful.
      USER_DELETED_S : Bool;   // ‘1’ temporarily when a requested user delete was successful
      LOGON_ATTEMPT_FAILED_S : Bool;   // ‘1’ temporarily when a logon attempt failed.
      NO_XRAY_DOOR_OPEN_S : Bool;   // ‘1’ temporarily when no X-rays possible because doors are open.
      NO_OPP_INCOM_AIR_LOW_S : Bool;   // ‘1’ temporarily when no operation possible due to low air pressure.
      GLOBAL_ALARM_S : Bool;   // ‘1’ when any alarm is present. Cleared when all alarms are reset.
      OTI_COMMS_FAULT_S : Bool;   // ‘1’ when comms fault between OTI and cRIO.
      LOCAL_REMOTE_S : Bool;   // ‘1’ when machine is in Remote mode
      MAINTENANCE_MODE_S : Bool;   // ‘1’ when in Maintenance Mode
      INCOM_AIR_PRESS_LO_S : Bool;   // ‘1’ when incoming air pressure less than low setpoint i.e. 4.5 bar.
      INCOM_AIR_PRESS_LOLO_S : Bool;   // ‘1’ when incoming air pressure less than low low setpoint i.e. 4.0 bar.
      PROC_WATERFLOW_HIGH_S : Bool;   // ‘1’ when flow rate greater than flow set-point plus allowed deviation.
      PROC_WATERFLOW_LOW_S : Bool;   // ‘1’ when flow rate less than flow set-point minus allowed deviation.
      FEEDER_RUNNING_S : Bool;   // ‘1’ when feeder is running.
      REMOTE_DNSTRM_INTLK_S : Bool;   // ‘1’ when downstream interlock healthy from PLC.
      HOLD_STATE_S : Bool;   // ‘1’ when feeder is prevented from running in “Processing” due to process interlock, low air pressure etc.
      WAIT_STATE_S : Bool;   // ‘1’ when in “Processing” state.
      PURGED_STATE_S : Bool;   // ‘1’ when a purge cycle is successfully completed. Cleared when feeder is next started.
      EJECTION_RATE_WARN_S : Bool;   // ‘1’ when ejection rate exceeds warning level.
      EJECTION_RATE_ALARM_S : Bool;   // ‘1’ when ejection rate exceeded ejection rate alarm level.
      MACH_ESTOP_ACTIVE_S : Bool;   // ‘1’ when E-stop active.
      XRAY_COOLW_TEMP_FAULT_S : Bool;   // ‘1’ when X-ray cooling water temperature to high or too low fault detected.
      XRAY_COOLW_FLOW_FAULT_S : Bool;   // ‘1’ when cooling water flow low fault detected.
      PROC_WATER_FLOW_S : Bool;   // ‘1’ when process water flow too high or too low fault detected. (Wet machine only)
      FRONT_SIDE_PROC_DOOR_S : Bool;   // ‘1’ when front side door open.
      BACK_SIDE_PROC_DOOR_S : Bool;   // ‘1’ when back side door open.
      FEEDER_DOOR_S : Bool;   // ‘1’ when feeder door open.
      HOOD_S : Bool;   // ‘1’ when hood open.
      CONC_TRACER_DOOR_S : Bool;   // ‘1’ when concentrate tracer door open.
      TAILINGS_TRACER_DOOR_S : Bool;   // ‘1’ when tailings tracer door open.
      CONC_TRACER_TRAY_S : Bool;   // ‘1’ when concentrate tracer tray in position.
      TAILINGS_TRACER_TRAY_S : Bool;   // ‘1’ when tailings tracer tray in position.
      PLANT_INLET_CHUTE_S : Bool;   // ‘1’ when plant inlet not in position.
      INSPECTION_COVER_S : Bool;   // ‘1’ when inspection cover not in position.
      PLANT_CONC_CHUTE_S : Bool;   // ‘1’ when plant concentrate chute not in position.
      PLANT_TAILINGS_CHUTE_S : Bool;   // ‘1’ when plant tailings chute not in position.
      INTERN_CONC_CHUTE_S : Bool;   // ‘1’ when internal concentrate chute not in position.
      INTERN_TAILINGS_CHUTE_S : Bool;   // ‘1’ when internal tailings chute not in position.
      DUSTEXTRACT_FLOW_FLT_S : Bool;   // ‘1’ when dust extractor flow fault detected (Dry machine only)
      SURGE_ARRESTOR_FLT_S : Bool;   // ‘1’ when one or more surge arrestors on the electrical panel is faulty.
      DXM_XRAY_GEN_COMM_FLT_S : Bool;   // ‘1’ when no comms between cRIO and Spellman DXM X-ray generator.
      DXM_HV_ENABLED_S : Bool;   // ‘1’ when X-rays ON.
      DXM_INTERLOCK_CLOSED_S : Bool;   // ‘1’ when interlock on X-ray generator is healthy.
      DXM_PS_FLT_S : Bool;   // ‘1’ when X-ray generator power supply fault detected.
      STATUS_BYTE6_SPARE7 : Bool;   // Status Byte-6 Spare
      STATUS_BYTE7_SPARE0 : Bool;   // Status Byte-7 Spare
      STATUS_BYTE7_SPARE1 : Bool;   // Status Byte-7 Spare
      STATUS_BYTE7_SPARE2 : Bool;   // Status Byte-7 Spare
      STATUS_BYTE7_SPARE3 : Bool;   // Status Byte-7 Spare
      STATUS_BYTE7_SPARE4 : Bool;   // Status Byte-7 Spare
      STATUS_BYTE7_SPARE5 : Bool;   // Status Byte-7 Spare
      STATUS_BYTE7_SPARE6 : Bool;   // Status Byte-7 Spare
      STATUS_BYTE7_SPARE7 : Bool;   // Status Byte-7 Spare
      STATUS_BYTE8_SPARE0 : Bool;   // Status Byte-8 Spare
      STATUS_BYTE8_SPARE1 : Bool;   // Status Byte-8 Spare
      STATUS_BYTE8_SPARE2 : Bool;   // Status Byte-8 Spare
      STATUS_BYTE8_SPARE3 : Bool;   // Status Byte-8 Spare
      STATUS_BYTE8_SPARE4 : Bool;   // Status Byte-8 Spare
      STATUS_BYTE8_SPARE5 : Bool;   // Status Byte-8 Spare
      STATUS_BYTE8_SPARE6 : Bool;   // Status Byte-8 Spare
      STATUS_BYTE8_SPARE7 : Bool;   // Status Byte-8 Spare
      STATUS_BYTE9_SPARE0 : Bool;   // Status Byte-9 Spare
      STATUS_BYTE9_SPARE1 : Bool;   // Status Byte-9 Spare
      STATUS_BYTE9_SPARE2 : Bool;   // Status Byte-9 Spare
      STATUS_BYTE9_SPARE3 : Bool;   // Status Byte-9 Spare
      STATUS_BYTE9_SPARE4 : Bool;   // Status Byte-9 Spare
      STATUS_BYTE9_SPARE5 : Bool;   // Status Byte-9 Spare
      STATUS_BYTE9_SPARE6 : Bool;   // Status Byte-9 Spare
      STATUS_BYTE9_SPARE7 : Bool;   // Status Byte-9 Spare
      STATUS_BYTE10_SPARE0 : Bool;   // Status Byte-10 Spare
      STATUS_BYTE10_SPARE1 : Bool;   // Status Byte-10 Spare
      STATUS_BYTE10_SPARE2 : Bool;   // Status Byte-10 Spare
      STATUS_BYTE10_SPARE3 : Bool;   // Status Byte-10 Spare
      STATUS_BYTE10_SPARE4 : Bool;   // Status Byte-10 Spare
      STATUS_BYTE10_SPARE5 : Bool;   // Status Byte-10 Spare
      STATUS_BYTE10_SPARE6 : Bool;   // Status Byte-10 Spare
      STATUS_BYTE10_SPARE7 : Bool;   // Status Byte-10 Spare
      MACHINE_STATE_S : Byte;   // 0-Initializing, 1-Ready, 2-Purging, 3-Display, 4-Calibrating, 5-Checker Cycle, 6-Processing Ready, 7-Processing, 8-Transition, 9-Alarm.
      DXM_COMMS_FLT_A : Bool;   // ALARM: DXM Comms fault
      DXM_XRAY_STATE_A : Bool;   // ALARM: DXM X-ray state alarm
      DXM_INTERLOCK_FLT_A : Bool;   // ALARM: DXM Interlock fault
      DXM_PSU_FAULT_A : Bool;   // ALARM: DXM Power supply fault
      DXM_NOTIN_REM_MODE_A : Bool;   // ALARM: DXM Not in remote mode fault
      DXM_ARC_FLT_A : Bool;   // ALARM: DXM Arc fault
      DXM_OVER_TEMP_FLT_A : Bool;   // ALARM: DXM Over temperature fault
      DXM_OVER_VOLT_FLT_A : Bool;   // ALARM: DXM Over voltage fault
      DXM_UNDER_VOLT_FLT_A : Bool;   // ALARM: DXM Under voltage fault
      DXM_OVER_CURRENT_FLT_A : Bool;   // ALARM: DXM Over current fault
      DXM_UNDER_CURRENT_FLT_A : Bool;   // ALARM: DXM Under current fault
      DXM_MODEL_NUMB_FLT_A : Bool;   // ALARM: DXM Model number fault
      ASI_COMMS_FAULT_A : Bool;   // ALARM: ASI Comms fault
      ASI_MISSING_SLAVE_FLT_A : Bool;   // ALARM: ASI Missing slave fault
      ASI_DUPL_SLAVE_FLT_A : Bool;   // ALARM: ASI Duplicate slave fault
      ASI_UNAUTH_SLAVE_FLT_A : Bool;   // ALARM: ASI Unauthorised slave fault
      ASIBUS_VOLT_LO_A : Bool;   // ALARM: ASI Bus voltage less than 28Vdc
      ASI_PERIP_FLT_A : Bool;   // ALARM: ASI Peripheral fault
      ASIBUS_VOLTS_EARTH_FLT_A : Bool;   // ALARM: ASI Bus voltage earth fault
      CRIO_MPLC_COMMS_FAIL_A : Bool;   // ALARM: cRIO - Machine PLC Comms failure
      CRIO_CHAS_TEMP_TOOHIGH_A : Bool;   // ALARM: cRIO chassis temperature too high
      XRAYGEN_COMP_TEMPHIGH_A : Bool;   // ALARM: X-ray generator compartment temperature high
      FPGA_HEARTBEAT_ERR_A : Bool;   // ALARM: FPGA heartbeat error
      FPGA_MODE_ERR_A : Bool;   // ALARM: FPGA mode error
      EJECT_FIRE_RATE_A : Bool;   // ALARM: Ejector fire rate alarm
      FEED_RATE_A : Bool;   // ALARM: Feed rate alarm
      COOLWATER_TEMP_HIGH_A : Bool;   // ALARM: Cooling water temperature high
      COOLWATER_TEMP_LOW_A : Bool;   // ALARM: Cooling water temperature low
      COOLWATER_FLOW_LO_A : Bool;   // ALARM: Cooling water flow low
      PROCWATER_FLOW_LO_ERR_A : Bool;   // ALARM: Process water flow low error
      PROCWATER_FLOW_HI_ERR_A : Bool;   // ALARM: Process water flow high error
      INCOM_AIRPRESS_LO_A : Bool;   // ALARM: Incoming air pressure low
      CALJIG_NOT_EXTEND_FLT_A : Bool;   // ALARM: Calibration jig not extending fault
      CALJIG_NOT_RETRACT_FLT_A : Bool;   // ALARM: Calibration jig not retracting fault
      CALJIGDR_NOT_OPEN_FLT_A : Bool;   // ALARM: Calibration jig door not opening fault
      CALJIGDR_NOT_CLOS_FLT_A : Bool;   // ALARM: Calibration jig door not closing fault
      CALIB_DEV_ERR_A : Bool;   // ALARM: Calibration deviation error
      CHANNEL_DATA_ZERO_A : Bool;   // ALARM: Channel data zero
      EJECTOR_ERRORS_A : Bool;   // ALARM: Ejector error(s)
      FRONT_SIDE_DR_OPN_A : Bool;   // ALARM: Front side door open
      BACK_SIDE_DR_OPN_A : Bool;   // ALARM: Back side door open
      FEEDER_DOOR_OPN_A : Bool;   // ALARM: Feeder door open
      CONC_TRACERDR_OPN_A : Bool;   // ALARM: Concentrate tracer door open
      TAILS_TRACERDR_OPN_A : Bool;   // ALARM: Tailings tracer door open
      HOOD_OPEN_A : Bool;   // ALARM: Hood open
      P_INLET_CHTE_NOTINPOS_A : Bool;   // ALARM: Plant inlet chute not in position
      INSPEC_COVER_OPN_A : Bool;   // ALARM: Inspection cover open
      P_CONC_CHTE_NOTINPOS_A : Bool;   // ALARM: Plant concentrate chute not in position
      P_TAILS_CHTE_NOTINPOS_A : Bool;   // ALARM: Plant tailings chute not in position
      INTCONC_CHTE_NOTINPOS_A : Bool;   // ALARM: Internal concentrate chute not in position
      INTTAILS_CHTE_NOTINPOS_A : Bool;   // ALARM: Internal tailings chute not in position
      DUST_EXTRACT_FLOW_FLT_A : Bool;   // ALARM: Dust extractor flow fault
      GATE_POSITION_FLT_A : Bool;   // ALARM: Gate position fault
      MACH_ESTOP_PRESSED_A : Bool;   // ALARM: Machine E-Stop button pressed
      SURGE_ARREST_FLT_A : Bool;   // ALARM: Surge arrestor fault
      ASI_SAFETY_BRIDGE_MISS_A : Bool;   // ALARM: ASI Safety bridging plug missing
      ASI_ESTOP_CONT_FB_FLT_A : Bool;   // ALARM: ASI E-stop contactor feedback fault
      XRAY_CONT_FB_FLT_A : Bool;   // ALARM: X-ray contactors feedback fault
      TRACERTRAY_INPOS_REM_A : Bool;   // ALARM: Tracer tray/s in position in remote mode
      CALIBJIG_COVR_NOTINPOS_A : Bool;   // ALARM: Calibration jig cover not in position
      ASI_ESTOP_CONT_FAIL_A : Bool;   // ALARM: ASI E-stop contactor failure
      ASI_PROJSLV_FLT_A : Bool;   // ALARM: ASI Projected slaves’ fault
      ASI_PARAM_OUTP_FLT_A : Bool;   // ALARM: ASI Parameter output fault
      ASISAFE_DEV_CODE_FLT_A : Bool;   // ALARM: ASI Safety device code fault
      "ASISAFE_PLC COMM_FLT_A" : Bool;   // ALARM: ASI Safety PLC comms alarm
      ASIBUS_VOLT_ASSYM_A : Bool;   // ALARM: ASi Bus voltage asymmetrical
      FILMW_EMPTY_FLT_A : Bool;   // ALARM: Film Winder empty fault
      FILMW_TORN_FLT_A : Bool;   // ALARM: Film Winder torn fault
      FILMW_NOTROT_FLT_A : Bool;   // ALARM: Film Winder not rotating fault
      FILMW_TIMOUT_A : Bool;   // ALARM: Film Winder timeout
      FILMW_COM_TIMOUT_FLT_A : Bool;   // ALARM: Film Winder comms timeout fault
      FILMWIND_MOT_A : Bool;   // ALARM: Film Winder motor alarm
      FILMWIND_UNKN_FLT_A : Bool;   // ALARM: Film Winder unknown fault
      DXM_KV_DEV_FLT_A : Bool;   // ALARM: DXM KV deviation fault
      DXM_MA_DEV_FLT_A : Bool;   // ALARM: DXM mA deviation fault
      ASI_SOFTW_NUM_FLT_A : Bool;   // ALARM: AS-i Software Number fault
      ALARM_BYTE10_SPARE4 : Bool;   // Alarm Byte-10 Spare
      ALARM_BYTE10_SPARE5 : Bool;   // Alarm Byte-10 Spare
      ALARM_BYTE10_SPARE6 : Bool;   // Alarm Byte-10 Spare
      ALARM_BYTE10_SPARE7 : Bool;   // Alarm Byte-10 Spare
      ALARM_BYTE11_SPARE0 : Bool;   // Alarm Byte-11 Spare
      ALARM_BYTE11_SPARE1 : Bool;   // Alarm Byte-11 Spare
      ALARM_BYTE11_SPARE2 : Bool;   // Alarm Byte-11 Spare
      ALARM_BYTE11_SPARE3 : Bool;   // Alarm Byte-11 Spare
      ALARM_BYTE11_SPARE4 : Bool;   // Alarm Byte-11 Spare
      ALARM_BYTE11_SPARE5 : Bool;   // Alarm Byte-11 Spare
      ALARM_BYTE11_SPARE6 : Bool;   // Alarm Byte-11 Spare
      ALARM_BYTE11_SPARE7 : Bool;   // Alarm Byte-11 Spare
      RECPAR_EJ_DELTIME_ACT : Byte;   // Recipe Parameter: Ejector Delay Time Actual, (0 to 50ms)
      RECPAR_EJ_ONTIME_ACT : Byte;   // Recipe Parameter: Ejection On Time Actual, (1 to 50ms)
      RECPAR_BLINT_TH_ACT : Word;   // Recipe Parameter: Algorithm Blue Intensity Threshold Actual, (60 to 10000mV)
      RECPAR_BLRD_OFF_ACT : Word;   // Recipe Parameter: Algorithm Blue-Red Discrimination Offset Actual, (0 to 10000)
      RECPAR_BLRD_RAT_ACT : Word;   // Recipe Parameter: Algorithm Blue-Red Discrimination Ratio Actual, (1 to 1000 equiv. 0.01 to 10.00)
      RECPAR_VIBFEED_SP_ACT : Byte;   // Recipe Parameter: Vibratory Feeder Setpoint Actual, (0 to 100%)
      RECPAR_AUTFEEDC_ACT : Bool;   // Recipe Parameter: Automatic Feeder Control Actual, OFF(0) – No closed loop control, ON(1) – Closed loop control
      RECPAR_RESERVED1 : Bool;   // Recipe Parameter: Reserved - Do Not Use
      RECPAR_RESERVED2 : Bool;   // Recipe Parameter: Reserved - Do Not Use
      RECPAR_RESERVED3 : Bool;   // Recipe Parameter: Reserved - Do Not Use
      RECPAR_RESERVED4 : Bool;   // Recipe Parameter: Reserved - Do Not Use
      RECPAR_RESERVED5 : Bool;   // Recipe Parameter: Reserved - Do Not Use
      RECPAR_RESERVED6 : Bool;   // Recipe Parameter: Reserved - Do Not Use
      RECPAR_RESERVED7 : Bool;   // Recipe Parameter: Reserved - Do Not Use
      RECPAR_GATEPOS_ACT : Byte;   // Recipe Parameter: Gate Position Actual - ‘0’ - No auto gate, ‘1’ - Gate in position 1(-2 +1mm), ‘2’ – Gate in position 2(-4+2mm), ‘3’ – Gate in position 3(-8+4mm), ‘4’ – Gate in position 4(-16+8mm), ‘5’ – Gate in position 5(-32+16mm)
      SPARE0 : Byte;   // Spare
      SPARE1 : DWord;   // Spare
      SPARE2 : DWord;   // Spare
      SPARE3 : DWord;   // Spare
      XRAY_KV_DEMAND_ACT : Byte;   // X-ray kV demand actual. U8. Expected range 0 to 40kV
      XRAY_MA_DEMAND_ACT : Byte;   // X-ray mA demand actual. U8. Expected range 0 to 23mA
      CCYCLE_REP_ACT : Byte;   // Checker Cycle repetitions actual. U8. Expected range 0 to 50%
      CALIBRATION_DEV_ACT : Byte;   // Calibration deviation actual. U8. Expected range 0 to 8
      EJE_RATE_WARN_LVL_ACT : Byte;   // Ejector rate warning level actual. U8. Expected range 0 to 20Ej/sec
      EJE_RATE_ALM_LVL_ACT : Byte;   // Ejector rate alarm level actual. U8. Expected range 0 to 20Ej/sec
      BLUE_CALIB_REF_ACT : Word;   // Blue calibration reference actual. U16.Expected range 0 to 0 to 10000mV
      RED_CALIB_REF_ACT : Word;   // Red calibration reference actual. U16.Expected range 0 to 0 to 10000mV
      PROC_WAT_FLOW_ALM_SP_ACT : Byte;   // Process water flow alarm setpoint actual. U8. Expected range 0 to 40litres/min
      PROC_WAT_FLOW_ALM_LVL_DEV_ACT : Byte;   // Process water flow alarm level deviation actual. U8. Expected range 0 to 10litres/min
      OVERRIDE_AUD_ALM_ACT : Bool;   // Override Audible Alarm Actual - Updated only on Change. ‘0’ – Not overridden, ‘1’ – Overridden
      OVERRIDE_EJE_ALM_ACT : Bool;   // Override Ejector Sense Feedback Alarms Actual - Updated only on Change. ‘0’ – Not overridden, ‘1’ – Overridden
      OVERRIDE_CCYCLE_SEQ_ACT : Bool;   // Override Checker Cycle Sequence Actual - Updated only on Change. ‘0’ – Not overridden, ‘1’ – Overridden
      MACHINE_TYPE_ACT : Bool;   // Machine Type Configured on the cRIO Actual - 1 = Dry 0 = Wet
      DETECTION_TYPE_ACT : Bool;   // Machine Detection Type Configured on cRIO Actual - 1 = Dual 0 = Single
      FILM_WINDER_ACT : Bool;   // Film Winder Actual. Dry machine only. '0' - Machine has no film winder, '1' - Machine has a film winder.
      SPARE4 : Bool;   // Spare
      SPARE5 : Bool;   // Spare
      CALIB_DEV_ALM_ENBL_CNT : Byte;   // Calibration deviation alarm enable count. U8. Expected range 0 to 8
      SIZEBLU_PMTSETP_ACT_ARR : DWord;   // Size of Blue PMT HV set-point actual array. U32. Expect value of 8 elements in array
      BLUPMT_HVSETP_ACT : Array[0..7] of Word;   // Blue PMT HV set-point actual. U16[8]. 8 x WORD corresponding to PMT1…PMT8. Expected range 0 to 1200V
      SIZERED_PMTSETP_ACT_ARR : DWord;   // Size of Red PMT HV set-point actual array. U32. Expect value of 8 elements in array
      REDPMT_HVSETP_ACT : Array[0..7] of Word;   // Red PMT HV set-point actual. U16[8]. 8 x WORD corresponding to PMT1…PMT8. Expected range 0 to 1200V
      SIZEBLU_PMTFDBK_ACT_ARR : DWord;   // Size of Blue PMT feedback multiplier actual array. U32. Expect value of 8 elements in array
      BLUPMT_HVFDBK_ACT : Array[0..7] of Byte;   // Holds the multiplier value for each blue channel PMT feedback signal: 0 – X1, 1 – X2, 2 – X10, 3 – X50.
      SIZERED_PMTFDBK_ACT_ARR : DWord;   // Size of Blue PMT feedback multiplier actual array. U32. Expect value of 8 elements in array
      REDPMT_HVFDBK_ACT : Array[0..7] of Byte;   // Holds the multiplier value for each red channel PMT feedback signal: 0 – X1, 1 – X2, 2 – X10, 3 – X50.
      SPARE6 : DWord;   // Spare
      SPARE7 : DWord;   // Spare
      SPARE8 : DWord;   // Spare
      SPARE9 : DWord;   // Spare
      SPARE10 : DWord;   // Spare
      SPARE11 : Word;   // Spare
      COOLWAT_FLOW_RATE : Byte;   // Cooling water flow rate. U8. Sensor feedback. Expected range 0 to 20 litres/min.
      COOLWAT_TEMP : Byte;   // Cooling water temperature. U8. Sensor feedback. Expected range 0 to 100⁰C.
      INCOM_AIR_PRESS : Word;   // Incoming air pressure. U16. Sensor feedback. Expected range 0 to 1000 which equates to 0 to 10.00bar.
      PROCWAT_FLOW_RATE : Word;   // Process water flow rate. U16. Sensor feedback. Expected range 0 to 4500 which equates to 0 to 45.00 litres/min. (Wet machine only)
      XRAY_GEN_COMP_TEMP : Byte;   // X-ray generator compartment temperature. U8. Sensor feedback. Expected range 0 to 100⁰C.
      XRAY_KV_FEEDBK : Byte;   // X-ray kV feedback. U8. X-ray feedback. Expected range 0 to 60kV.
      XRAY_MA_FEEDBK : Byte;   // X-ray mA feedback. U8. X-ray feedback. Expected range 0 to 25mA.
      HEARTBEAT_RTSYS_MPLC : Byte;   // Communications heartbeat from Machine Controller.
      LOOKUP_TABLE_USER_NAME : Array[0..7] of Byte;   // Lookup table username. Username at requested security lookup table pointer, 8-character string
      LOOKUP_TABLE_ACCESS_LVL : Byte;   // Lookup table access level. Access level at requested security lookup table pointer
      LOGGED_ON_USER_ACCES_LVL : Byte;   // Access level for the current logged on user: 0-Operator (default)1-Technician2-Metallurgist 3-Administrator
      CURRENT_USER_NAME : Array[0..7] of Byte;   // Current User Name Logged On to the cRIO, 8 character string
      VIB_FEED_FEEDBK : Byte;   // Vibratory feeder feedback. U8. Feeder feedback. Expected range 0 to 100% full scale deflection.
      GATE_POS_ACT : Byte;   // Reflects the current/actual position of the Auto gate if present. ‘0’ - No auto gate, '1’ – gate at position1(-2 +1mm), '2’ – gate at position2(-4 +2mm), '3’ – Gate at position3(-8 +4mm), '4’ – Gate at position4(-16 +8mm), '5’ – Gate at position5(-32 +16mm)
      RESERVED_UP_REC_CMMD : Byte;   // Remote_Recipe_Update_Reserved_for_Controller_and_PLC
      CRIO_CONT_TIME_HRS : Byte;   // System time - hours: 0 - 23
      CRIO_CONT_TIME_MINS : Byte;   // System time - minutes: 0 - 59
      CRIO_CONT_TIME_SECS : Byte;   // System time - seconds: 0 - 59
      CRIO_CONT_TIME_CEN : Byte;   // System date - centuary : 0 - 99
      CRIO_CONT_TIME_YRS : Byte;   // System date - year: 0 - 99
      CRIO_CONT_TIME_MNT : Byte;   // System date - month: 1-12
      CRIO_CONT_TIME_DAY : Byte;   // System date - day: 1-31
      MACH_POWER_CONSUMP : DWord;   // U32. Running total of power consumption in kWh of the machine.
      MACH_PROCWATER_CONSUMP : DWord;   // U32. Running total process water consumption in kilo litres of the machine.
      FEEDER_STOPPED_STATUS : Byte;   // Reason why feeder is not running in Processing state or feeder cannot be started in Processing Ready state.Reason why feeder is not running in Processing state or feeder cannot be started in Processing Ready state. 0 – none (feeder is running or can be started); 1 – Processing water flow low; 2 – Incoming air pressure low low; 3 – Ejection rate alarm; 4 – Downstream interlock
      SPARE12 : Byte;   // Spare
      SPARE13 : DWord;   // Spare
      SPARE14 : DWord;   // Spare
      SPARE15 : DWord;   // Spare
      BLUE_PEAK_INTEN : Word;   // Blue Peak Intensity. U16. Holds blue value of last detection. Expected range 0 to 10000mV
      RED_PEAK_INTEN : Word;   // Red Peak Intensity. U16. Holds red value of last peak detection. Expected range 0 to 10000mV
      MOST_ACTIVE_FIRE_CHAN : Byte;   // Most active fire rate channel. U8. Indicates the channel that currently has the highest firing rate. Expected range 0 to 8
      MOST_ACTIVE_CHAN_FIRE : Byte;   // Most active channel firing rate. U8. Indicates the most active channels firing rate [ej/sec] multiplied by 10 i.e. 225 received therefore indicates 22.5 ej/sec
      LAST_EJECT_ACTIV : Byte;   // Last Ejector Activated. Indicates the channel of the last ejector activated. Expected range 0 to 8
      SPARE16 : Byte;   // Spare
      RES_NUMELEM_IN_ARRAY_0 : DWord;   // Reserved (Holds number of elements in array)
      EJECT_DELAY_RESP : Array[0..15] of Byte;   // 16 x BYTE corresponding to CH1_1…CH8_2. Expected range 0 to 255
      RES_NUMELEM_IN_ARRAY_1 : DWord;   // Reserved (Holds number of elements in array)
      EJECT_DUR_RESP : Array[0..15] of Byte;   // 16 x BYTE corresponding to CH1_1…CH8_2. Expected range 0 to 255
      RES_NUMELEM_IN_ARRAY_2 : DWord;   // Reserved (Holds number of elements in array)
      EJECT_ERROR_HIST : Array[0..15] of DWord;   // 16 x DWORD corresponding to CH1_1…CH8_2 (64 bytes)
      RES_NUMELEM_IN_ARRAY_3 : DWord;   // Reserved (Holds number of elements in array)
      EJECT_PROFILE : Array[0..7] of DWord;   // 8 x DWORD corresponding to CH1…CH8 (32 bytes)
      RES_NUMELEM_IN_ARRAY_4 : DWord;   // Reserved (Holds number of elements in array)
      ACCEP_PROFILE : Array[0..7] of DWord;   // 8 x DWORD corresponding to CH1…CH8 (32 bytes)
      RES_NUMELEM_IN_ARRAY_5 : DWord;   // Reserved (Holds number of elements in array)
      REJECT_PROFILE : Array[0..7] of DWord;   // 8 x DWORD corresponding to CH1…CH8 (32 bytes)
      RES_NUMELEM_IN_ARRAY_6 : DWord;   // Reserved (Holds number of elements in array)
      BLUE_CALIB_REF_DATA : Array[0..7] of Word;   // 8 x WORD corresponding to CH1…CH8 (16 bytes)
      RES_NUMELEM_IN_ARRAY_7 : DWord;   // Reserved (Holds number of elements in array)
      BLUE_CALIB_CC_DATA : Array[0..7] of Word;   // 8 x WORD corresponding to CH1…CH8 (16 bytes)
      RES_NUMELEM_IN_ARRAY_8 : DWord;   // Reserved (Holds number of elements in array)
      RED_CALIB_REF_DATA : Array[0..7] of Word;   // 8 x WORD corresponding to CH1…CH8 (16 bytes)
      RES_NUMELEM_IN_ARRAY_9 : DWord;   // Reserved (Holds number of elements in array)
      RED_CALIB_CC_DATA : Array[0..7] of Word;   // 8 x WORD corresponding to CH1…CH8 (16 bytes)
      RES_NUMELEM_IN_ARRAY_10 : DWord;   // Reserved (Holds number of elements in array)
      ACCEPT_LI_HIST : Array[0..63] of DWord;   // 64 x DWORD corresponding to bin no 1…64 (256 bytes)
      RES_NUMELEM_IN_ARRAY_11 : DWord;   // Reserved (Holds number of elements in array)
      REJECT_LI_HIST : Array[0..63] of DWord;   // 64 x DWORD corresponding to bin no 1…64 (256 bytes)
      RES_NUMELEM_IN_ARRAY_12 : DWord;   // Reserved (Holds number of elements in array)
      RED_LI_HIST : Array[0..63] of DWord;   // 64 x DWORD corresponding to bin no 1…64 (256 bytes)
      RES_NUMELEM_IN_ARRAY_13 : DWord;   // Reserved (Holds number of elements in array)
      BLUE_RED_RATIO_LI_HIST : Array[0..63] of DWord;   // 64 x DWORD corresponding to bin no 1…64 (256 bytes)
      LI_HIST_CLR_TIME_HRS : Byte;   // LI histogram clear time - hours: 0 - 23
      LI_HIST_CLR_TIME_MINS : Byte;   // LI histogram clear time - minutes: 0 - 59
      LI_HIST_CLR_TIME_SECS : Byte;   // LI histogram clear time - seconds: 0 - 59
      LI_HIST_CLR_DATE_CENT : Byte;   // LI histogram clear date - centuary : 0 - 99
      LI_HIST_CLR_DATE_YRS : Byte;   // LI histogram clear date - year: 0 - 99
      LI_HIST_CLR_DATE_MNT : Byte;   // LI histogram clear date - month: 1-12
      LI_HIST_CLR_DATE_DAY : Byte;   // LI histogram clear date - day: 1-31
      SPARE17 : Byte;   // Spare
      TIME_SINCE_HIST_CLR : DWord;   // DWORD indicating the time difference between the Current Time and the Histogram Clear Time, in seconds
      SPARE18 : DWord;   // Spare
      SPARE19 : DWord;   // Spare
      SPARE20 : DWord;   // Spare
      SPARE21 : DWord;   // Spare
      SPARE22 : DWord;   // Spare
      SPARE23 : DWord;   // Spare
   END_STRUCT;
END_TYPE

TYPE "118MK2_PlantIF_Cmd"
// stored: IsFailsafeCompliant false
   STRUCT
      Start_M_PCS { ExternalAccessible := 'False'; ExternalVisible := 'False'; ExternalWritable := 'False'} : Bool;   // Moves machine to Processing Material State. Feeder is not started.
      Stop_M_PCS { ExternalAccessible := 'False'; ExternalVisible := 'False'; ExternalWritable := 'False'} : Bool;   // Moves machine to Standby State. Hence also used to exit Display mode.
      Start_Feeding_M_PCS { ExternalAccessible := 'False'; ExternalVisible := 'False'; ExternalWritable := 'False'} : Bool;   // Starts the vibratory feeder
      Stop_Feeding_M_PCS { ExternalAccessible := 'False'; ExternalVisible := 'False'; ExternalWritable := 'False'} : Bool;   // Stops the vibratory feeder
      Checker_Cycle_M_PCS { ExternalAccessible := 'False'; ExternalVisible := 'False'; ExternalWritable := 'False'} : Bool;   // Initiates a Checker Cycle sequence
      Purge_M_PCS { ExternalAccessible := 'False'; ExternalVisible := 'False'; ExternalWritable := 'False'} : Bool;   // Initiates a material purge sequence
      Acknowledge_Alarm_PCS { ExternalAccessible := 'False'; ExternalVisible := 'False'; ExternalWritable := 'False'} : Bool;   // Acknowledges asserted alarm/s. Siren is deactivated.
      Reset_Alarm_PCS { ExternalAccessible := 'False'; ExternalVisible := 'False'; ExternalWritable := 'False'} : Bool;   // Resets asserted alarm/s
      Manual_Req_PCS { ExternalAccessible := 'False'; ExternalVisible := 'False'; ExternalWritable := 'False'} : Bool;   // Initiates a Mode Request, Toggles between Manual/Auto
      Calibrate_M_PCS { ExternalAccessible := 'False'; ExternalVisible := 'False'; ExternalWritable := 'False'} : Bool;   // Automatically adjusts the PMT HV setpoints to achieve the desired calibration reference
      Display_M_PCS { ExternalAccessible := 'False'; ExternalVisible := 'False'; ExternalWritable := 'False'} : Bool;   // Moves machine to Display state where blue and red channel data for all 8 channels is acquired every 250ms
      Save_As_Reference_PCS { ExternalAccessible := 'False'; ExternalVisible := 'False'; ExternalWritable := 'False'} : Bool;   // Saves the most recent calibration data for both the blue and red channels as the reference curve in the RT Controller non-volatile memory
      Save_Oper_Params_PCS { ExternalAccessible := 'False'; ExternalVisible := 'False'; ExternalWritable := 'False'} : Bool;   // Saves all operation parameters to NVM on the RT Controller
      Upd_Sys_DateTime_PCS { ExternalAccessible := 'False'; ExternalVisible := 'False'; ExternalWritable := 'False'} : Bool;   // Issue a System Date and Time Update
      Spare6 { ExternalAccessible := 'False'; ExternalVisible := 'False'; ExternalWritable := 'False'} : Bool;   // Spare
      Spare7 { ExternalAccessible := 'False'; ExternalVisible := 'False'; ExternalWritable := 'False'} : Bool;   // Spare
      Clr_LiHist_M_PCS { ExternalAccessible := 'False'; ExternalVisible := 'False'; ExternalWritable := 'False'} : Bool;   // Clears Accepted, Rejected, Red and Blue-Red Ratio Luminescence Intensity Histograms
      Clr_Profile_M_PCS { ExternalAccessible := 'False'; ExternalVisible := 'False'; ExternalWritable := 'False'} : Bool;   // Clears ejection, accepted & rejected profiles
      Clr_EjecErrHist_M_PCS { ExternalAccessible := 'False'; ExternalVisible := 'False'; ExternalWritable := 'False'} : Bool;   // Resets all the data values in the Ejector error histograms to zero
      Clr_EjecResProf_M_PCS { ExternalAccessible := 'False'; ExternalVisible := 'False'; ExternalWritable := 'False'} : Bool;   // Clears ejector delay response and ejector duration response profiles
      Clr_CCCalData_M_PCS { ExternalAccessible := 'False'; ExternalVisible := 'False'; ExternalWritable := 'False'} : Bool;   // Clears Blue and Red Checker cycle calibration data profiles
      Spare8 { ExternalAccessible := 'False'; ExternalVisible := 'False'; ExternalWritable := 'False'} : Bool;   // Spare
      Spare9 { ExternalAccessible := 'False'; ExternalVisible := 'False'; ExternalWritable := 'False'} : Bool;   // Spare
      Spare10 { ExternalAccessible := 'False'; ExternalVisible := 'False'; ExternalWritable := 'False'} : Bool;   // Spare
      Spare11 { ExternalAccessible := 'False'; ExternalVisible := 'False'; ExternalWritable := 'False'} : Bool;   // Spare
      Spare12 { ExternalAccessible := 'False'; ExternalVisible := 'False'; ExternalWritable := 'False'} : Bool;   // Spare
      Spare13 { ExternalAccessible := 'False'; ExternalVisible := 'False'; ExternalWritable := 'False'} : Bool;   // Spare
      Spare14 { ExternalAccessible := 'False'; ExternalVisible := 'False'; ExternalWritable := 'False'} : Bool;   // Spare
      Spare15 { ExternalAccessible := 'False'; ExternalVisible := 'False'; ExternalWritable := 'False'} : Bool;   // Spare
      Spare16 { ExternalAccessible := 'False'; ExternalVisible := 'False'; ExternalWritable := 'False'} : Bool;   // Spare
      Spare17 { ExternalAccessible := 'False'; ExternalVisible := 'False'; ExternalWritable := 'False'} : Bool;   // Spare
      Spare18 { ExternalAccessible := 'False'; ExternalVisible := 'False'; ExternalWritable := 'False'} : Bool;   // Spare
      Add_New_User_PCS { ExternalAccessible := 'False'; ExternalVisible := 'False'; ExternalWritable := 'False'} : Bool;   // Adds a new User based Username, password and Access level
      Del_Select_User_PCS { ExternalAccessible := 'False'; ExternalVisible := 'False'; ExternalWritable := 'False'} : Bool;   // Delete the user specified by the current lookup table pointer, from the cRIO security lookup table
      Logon_User_PCS { ExternalAccessible := 'False'; ExternalVisible := 'False'; ExternalWritable := 'False'} : Bool;   // Authorise user based on the specified username and password - the cRIO would return the appropriate access level
      LogOff_User_PCS { ExternalAccessible := 'False'; ExternalVisible := 'False'; ExternalWritable := 'False'} : Bool;   // Log off user – the Access Level of 0 would return after command
      Change_User_Pass_PCS { ExternalAccessible := 'False'; ExternalVisible := 'False'; ExternalWritable := 'False'} : Bool;   // Change password for currently logged on user as specified in “User password”
      Lookup_User_PCS { ExternalAccessible := 'False'; ExternalVisible := 'False'; ExternalWritable := 'False'} : Bool;   // Retrieve the Username and Access Level at the specified Sec. Lookup table pntr
      Spare19 { ExternalAccessible := 'False'; ExternalVisible := 'False'; ExternalWritable := 'False'} : Bool;   // Spare
      Spare20 { ExternalAccessible := 'False'; ExternalVisible := 'False'; ExternalWritable := 'False'} : Bool;   // Spare
      Start_A_PCS { ExternalAccessible := 'False'; ExternalVisible := 'False'; ExternalWritable := 'False'} : Bool;   // Sequencer Start
      Stop_A_PCS { ExternalAccessible := 'False'; ExternalVisible := 'False'; ExternalWritable := 'False'} : Bool;   // Sequencer Stop
      Start_Feeding_A_PCS { ExternalAccessible := 'False'; ExternalVisible := 'False'; ExternalWritable := 'False'} : Bool;   // Sequencer Feeder Start
      Stop_Feeding_A_PCS { ExternalAccessible := 'False'; ExternalVisible := 'False'; ExternalWritable := 'False'} : Bool;   // Sequencer Feeder Stop
      Checker_Cycle_A_PCS { ExternalAccessible := 'False'; ExternalVisible := 'False'; ExternalWritable := 'False'} : Bool;   // Sequencer Checker Cycle Req
      Purge_A_PCS { ExternalAccessible := 'False'; ExternalVisible := 'False'; ExternalWritable := 'False'} : Bool;   // Sequencer Purge Req
      Spare21 { ExternalAccessible := 'False'; ExternalVisible := 'False'; ExternalWritable := 'False'} : Bool;   // Spare
      Spare22 { ExternalAccessible := 'False'; ExternalVisible := 'False'; ExternalWritable := 'False'} : Bool;   // Spare
      User_Name { ExternalAccessible := 'False'; ExternalVisible := 'False'; ExternalWritable := 'False'} : Array[0..7] of Byte;   // User Name for Authorization/addition on Machine lookup table
      User_Password { ExternalAccessible := 'False'; ExternalVisible := 'False'; ExternalWritable := 'False'} : Array[0..7] of Byte;   // User Password for Authorization/addition on Machine lookup table
      User_Access_Level { ExternalAccessible := 'False'; ExternalVisible := 'False'; ExternalWritable := 'False'} : Byte;   // User Access Level for Addintion on Machine Lookup table
      Sec_LookupTable_Pntr { ExternalAccessible := 'False'; ExternalVisible := 'False'; ExternalWritable := 'False'} : Byte := 16#0;   // Lookup user in security lookup table. Range: 1 to 40. 0 = hidden administrator.
      Save_Recipe { ExternalAccessible := 'False'; ExternalVisible := 'False'; ExternalWritable := 'False'} : Bool;   // 1 to Save Current Recipe
      Delete_Recipe { ExternalAccessible := 'False'; ExternalVisible := 'False'; ExternalWritable := 'False'} : Bool;   // 1 to Delete Current Recipe
      Copy_Recipe { ExternalAccessible := 'False'; ExternalVisible := 'False'; ExternalWritable := 'False'} : Bool;   // 1 to Copy a Recipe
      Spare23 { ExternalAccessible := 'False'; ExternalVisible := 'False'; ExternalWritable := 'False'} : Bool;   // Spare
      Spare24 { ExternalAccessible := 'False'; ExternalVisible := 'False'; ExternalWritable := 'False'} : Bool;   // Spare
      Spare25 { ExternalAccessible := 'False'; ExternalVisible := 'False'; ExternalWritable := 'False'} : Bool;   // Spare
      Spare26 { ExternalAccessible := 'False'; ExternalVisible := 'False'; ExternalWritable := 'False'} : Bool;   // Spare
      Spare27 { ExternalAccessible := 'False'; ExternalVisible := 'False'; ExternalWritable := 'False'} : Bool;   // Spare
      Select_Recipe_No { ExternalAccessible := 'False'; ExternalVisible := 'False'; ExternalWritable := 'False'} : Byte;   // Select Active Recipe
      Dest_Recipe_No { ExternalAccessible := 'False'; ExternalVisible := 'False'; ExternalWritable := 'False'} : Byte;   // Set the Destination Number to copy to
      Spare28 { ExternalAccessible := 'False'; ExternalVisible := 'False'; ExternalWritable := 'False'} : Byte;   // Spare
      ScratchPad { ExternalAccessible := 'False'; ExternalVisible := 'False'; ExternalWritable := 'False'} : "118MK2_RecipeEdit";   // Scratch Pad for Recipe Edits
      Remote_DSInlk_PCS { ExternalAccessible := 'False'; ExternalVisible := 'False'; ExternalWritable := 'False'} : Bool;   // Status of the D/S int. on either MachPLC-H/W or PlntPLC-S/W 0: Inlk 1: Healthy
      Remote_SpareCMD1_PCS { ExternalAccessible := 'False'; ExternalVisible := 'False'; ExternalWritable := 'False'} : Bool;   // Spare Remote Commands
      Remote_SpareCMD2_PCS { ExternalAccessible := 'False'; ExternalVisible := 'False'; ExternalWritable := 'False'} : Bool;   // Spare Remote Commands
      Remote_SpareCMD3_PCS { ExternalAccessible := 'False'; ExternalVisible := 'False'; ExternalWritable := 'False'} : Bool;   // Spare Remote Commands
      Remote_SpareCMD4_PCS { ExternalAccessible := 'False'; ExternalVisible := 'False'; ExternalWritable := 'False'} : Bool;   // Spare Remote Commands
      Remote_SpareCMD5_PCS { ExternalAccessible := 'False'; ExternalVisible := 'False'; ExternalWritable := 'False'} : Bool;   // Spare Remote Commands
      Remote_SpareCMD6_PCS { ExternalAccessible := 'False'; ExternalVisible := 'False'; ExternalWritable := 'False'} : Bool;   // Spare Remote Commands
      Remote_SpareCMD7_PCS { ExternalAccessible := 'False'; ExternalVisible := 'False'; ExternalWritable := 'False'} : Bool;   // Spare Remote Commands
      SOC_Authorization { ExternalAccessible := 'False'; ExternalVisible := 'False'; ExternalWritable := 'False'} : Bool;   // Supervised Operator Control Authorization, 0 = No Auth, 1 = Grant Auth
      SOC_Req_Acknowledge { ExternalAccessible := 'False'; ExternalVisible := 'False'; ExternalWritable := 'False'} : Bool;   // Plant acknowledgement of SOC request; 0 = not acknowledged, 1 = request acknowledged
      Spare30 { ExternalAccessible := 'False'; ExternalVisible := 'False'; ExternalWritable := 'False'} : Bool;   // Spare
      Spare31 { ExternalAccessible := 'False'; ExternalVisible := 'False'; ExternalWritable := 'False'} : Bool;   // Spare
      Spare32 { ExternalAccessible := 'False'; ExternalVisible := 'False'; ExternalWritable := 'False'} : Bool;   // Spare
      Spare33 { ExternalAccessible := 'False'; ExternalVisible := 'False'; ExternalWritable := 'False'} : Bool;   // Spare
      Spare34 { ExternalAccessible := 'False'; ExternalVisible := 'False'; ExternalWritable := 'False'} : Bool;   // Spare
      Spare35 { ExternalAccessible := 'False'; ExternalVisible := 'False'; ExternalWritable := 'False'} : Bool;   // Spare
      Heartbeat_PCS_MPLC { ExternalAccessible := 'False'; ExternalVisible := 'False'; ExternalWritable := 'False'} : Byte;   // Receive Comms Heartbeat from Plant PLC
      Spare36 { ExternalAccessible := 'False'; ExternalVisible := 'False'; ExternalWritable := 'False'} : Byte;   // Spare
      RTC_Update_PCS { ExternalAccessible := 'False'; ExternalVisible := 'False'; ExternalWritable := 'False'; S7_SetPoint := 'True'} : "RTC";   // Real Time Clock Update Data
      PCS_Data_Range { ExternalAccessible := 'False'; ExternalVisible := 'False'; ExternalWritable := 'False'} : Byte;   // Plant data range: 0 (default)= Basic command and statuses; 1=Include messages; 2=Include MAPCOM data
      Spare37 { ExternalAccessible := 'False'; ExternalVisible := 'False'; ExternalWritable := 'False'} : Byte;   // Spare
      Spare38 { ExternalAccessible := 'False'; ExternalVisible := 'False'; ExternalWritable := 'False'} : Word;   // Spare
      Spare39 { ExternalAccessible := 'False'; ExternalVisible := 'False'; ExternalWritable := 'False'} : Word;   // End of Receive Data Structure - 70 Bytes
   END_STRUCT;
END_TYPE

TYPE "118MK2_PlantIF_Cmd_OPC"
// stored: IsFailsafeCompliant false
   STRUCT
      Start_M_PCS : Bool;   // Moves machine to Processing Material State. Feeder is not started.
      Stop_M_PCS : Bool;   // Moves machine to Standby State. Hence also used to exit Display mode.
      Start_Feeding_M_PCS : Bool;   // Starts the vibratory feeder
      Stop_Feeding_M_PCS : Bool;   // Stops the vibratory feeder
      Checker_Cycle_M_PCS : Bool;   // Initiates a Checker Cycle sequence
      Purge_M_PCS : Bool;   // Initiates a material purge sequence
      Acknowledge_Alarm_PCS : Bool;   // Acknowledges asserted alarm/s. Siren is deactivated.
      Reset_Alarm_PCS : Bool;   // Resets asserted alarm/s
      Manual_Req_PCS : Bool;   // Initiates a Mode Request, Toggles between Manual/Auto
      Calibrate_M_PCS : Bool;   // Automatically adjusts the PMT HV setpoints to achieve the desired calibration reference
      Display_M_PCS : Bool;   // Moves machine to Display state where blue and red channel data for all 8 channels is acquired every 250ms
      Save_As_Reference_PCS : Bool;   // Saves the most recent calibration data for both the blue and red channels as the reference curve in the RT Controller non-volatile memory
      Save_Oper_Params_PCS : Bool;   // Saves all operation parameters to NVM on the RT Controller
      Upd_Sys_DateTime_PCS : Bool;   // Issue a System Date and Time Update
      Spare6 : Bool;   // Spare
      Spare7 : Bool;   // Spare
      Clr_LiHist_M_PCS : Bool;   // Clears Accepted, Rejected, Red and Blue-Red Ratio Luminescence Intensity Histograms
      Clr_Profile_M_PCS : Bool;   // Clears ejection, accepted & rejected profiles
      Clr_EjecErrHist_M_PCS : Bool;   // Resets all the data values in the Ejector error histograms to zero
      Clr_EjecResProf_M_PCS : Bool;   // Clears ejector delay response and ejector duration response profiles
      Clr_CCCalData_M_PCS : Bool;   // Clears Blue and Red Checker cycle calibration data profiles
      Spare8 : Bool;   // Spare
      Spare9 : Bool;   // Spare
      Spare10 : Bool;   // Spare
      Spare11 : Bool;   // Spare
      Spare12 : Bool;   // Spare
      Spare13 : Bool;   // Spare
      Spare14 : Bool;   // Spare
      Spare15 : Bool;   // Spare
      Spare16 : Bool;   // Spare
      Spare17 : Bool;   // Spare
      Spare18 : Bool;   // Spare
      Add_New_User_PCS : Bool;   // Adds a new User based Username, password and Access level
      Del_Select_User_PCS : Bool;   // Delete the user specified by the current lookup table pointer, from the cRIO security lookup table
      Logon_User_PCS : Bool;   // Authorise user based on the specified username and password - the cRIO would return the appropriate access level
      LogOff_User_PCS : Bool;   // Log off user – the Access Level of 0 would return after command
      Change_User_Pass_PCS : Bool;   // Change password for currently logged on user as specified in “User password”
      Lookup_User_PCS : Bool;   // Retrieve the Username and Access Level at the specified Sec. Lookup table pntr
      Spare19 : Bool;   // Spare
      Spare20 : Bool;   // Spare
      Start_A_PCS : Bool;   // Sequencer Start
      Stop_A_PCS : Bool;   // Sequencer Stop
      Start_Feeding_A_PCS : Bool;   // Sequencer Feeder Start
      Stop_Feeding_A_PCS : Bool;   // Sequencer Feeder Stop
      Checker_Cycle_A_PCS : Bool;   // Sequencer Checker Cycle Req
      Purge_A_PCS : Bool;   // Sequencer Purge Req
      Spare21 : Bool;   // Spare
      Spare22 : Bool;   // Spare
      User_Name : Array[0..7] of Byte;   // User Name for Authorization/addition on Machine lookup table
      User_Password : Array[0..7] of Byte;   // User Password for Authorization/addition on Machine lookup table
      User_Access_Level : Byte;   // User Access Level for Addintion on Machine Lookup table
      Sec_LookupTable_Pntr : Byte := 16#0;   // Lookup user in security lookup table. Range: 1 to 40. 0 = hidden administrator.
      Save_Recipe : Bool;   // 1 to Save Current Recipe
      Delete_Recipe : Bool;   // 1 to Delete Current Recipe
      Copy_Recipe : Bool;   // 1 to Copy a Recipe
      Spare23 : Bool;   // Spare
      Spare24 : Bool;   // Spare
      Spare25 : Bool;   // Spare
      Spare26 : Bool;   // Spare
      Spare27 : Bool;   // Spare
      Select_Recipe_No : Byte;   // Select Active Recipe
      Dest_Recipe_No : Byte;   // Set the Destination Number to copy to
      Spare28 : Byte;   // Spare
      ScratchPad : "118MK2_RecipeEdit";   // Scratch Pad for Recipe Edits
      Remote_DSInlk_PCS : Bool;   // Status of the D/S int. on either MachPLC-H/W or PlntPLC-S/W 0: Inlk 1: Healthy
      Remote_SpareCMD1_PCS : Bool;   // Spare Remote Commands
      Remote_SpareCMD2_PCS : Bool;   // Spare Remote Commands
      Remote_SpareCMD3_PCS : Bool;   // Spare Remote Commands
      Remote_SpareCMD4_PCS : Bool;   // Spare Remote Commands
      Remote_SpareCMD5_PCS : Bool;   // Spare Remote Commands
      Remote_SpareCMD6_PCS : Bool;   // Spare Remote Commands
      Remote_SpareCMD7_PCS : Bool;   // Spare Remote Commands
      SOC_Authorization : Bool;   // Supervised Operator Control Authorization, 0 = No Auth, 1 = Grant Auth
      SOC_Req_Acknowledge : Bool;   // Spare
      Spare30 : Bool;   // Spare
      Spare31 : Bool;   // Spare
      Spare32 : Bool;   // Spare
      Spare33 : Bool;   // Spare
      Spare34 : Bool;   // Spare
      Spare35 : Bool;   // Spare
      Heartbeat_PCS_MPLC : Byte;   // Receive Comms Heartbeat from Plant PLC
      Spare36 : Byte;   // Spare
      RTC_Update_PCS { S7_SetPoint := 'True'} : "RTC";   // Real Time Clock Update Data
      PCS_Data_Range : Byte;   // Plant data range: 0 (default)= Basic command and statuses; 1=Include messages; 2=Include MAPCOM data
      Spare37 : Byte;   // Spare
      Spare38 : Word;   // Spare
      Spare39 : Word;   // End of Receive Data Structure - 70 Bytes
   END_STRUCT;
END_TYPE

TYPE "118MK2_PlantIF_Status"
// stored: IsFailsafeCompliant false
   STRUCT
      PlantSeq_Data { S7_SetPoint := 'True'} : "PLANT_SEQ_STATE";
      Status_Data { S7_SetPoint := 'True'} : "118MK2_PlantData";   // Status Information from Machine
      Recipe_Data { S7_SetPoint := 'True'} : "118MK2_RecipeData";   // Recipe Information from Machine
   END_STRUCT;
END_TYPE

